				 FOR i:=1 TO gc_ModuleProNo BY 1 DO
						 MEMSET(ADR(tsModuleProcess[i]),0,SIZEOF(tsModuleProcess[i]));
				 END_FOR
			station.iStepAuto:= 20;
  	20://区分上料还是请料
			 IF  station.xEmptying  THEN
					station.iStepAuto:= 1000;
			 ELSIF station.xEmptyDone THEN
					  station.xDone:=TRUE;
						station.iStepAuto:= 0;
			 ELSE
					station.iStepAuto:= 30;
			 END_IF
		30://Restore_after_Estop_Process1-拍照流程
				IF  axBypassSignal[1] OR fbMachine[1].xTryRun THEN
						station.iStepAuto :=110 ;
				ELSE    
						station.iStepAuto :=40; 
				END_IF
		40://启动链板线
			tsModuleProcess[1].xProcessNotStarted:=TRUE;
			IF   NOT _FirstFlag[3] OR station.xSingleRunning THEN
					fbFlowLine.xIRunningPremit:=TRUE;
			END_IF
				station.iStepAuto:=50;	
	 45://
				 fbFlowLine.xIRunningPremit:=TRUE;
				 station.iStepAuto:=46;	
	 46://判断是否需要拍照
				//IF  NOT	_FirstCycle[3] THEN
					 station.iStepAuto:=50;	
				//ELSE
				//	 station.iStepAuto:=80;
				// END_IF
	 50://Y轴去拍照位置
		 arTonDelay[03](IN:=FALSE);
		 fbYAxisMove.xMoveAuto[2]:=TRUE;
		 IF  fbYAxisMove.xMoveInPos[2] THEN
					station.iStepAuto:=60;	
		 END_IF
	60://等待链板线孔板到位 
			arTonDelay[03](IN:=TRUE , PT:=T#10S , Q=> , ET=> ); 
			IF 	fbFlowLine.xQDone  THEN
					 station.iStepAuto:=65;	
			ELSIF fbFlowLine.xQError OR  	arTonDelay[03].Q THEN
			 		arTonDelay[03](IN:=FALSE);
					fbFlowLine.xIInit:=TRUE;
					 station.iStepAuto:=45;	
					station.adwAlarm[1].31	:=	TRUE;//	S01上料工位-链板线运行超时,请复位
			END_IF
	65://链板线停止
				fbFlowLine.xIMotorStop :=TRUE;
			IF NOT  fbFlowLine.xQMotorStart THEN
			 			 station.iStepAuto:=70;	
			END_IF
	70://第一个循环相机拍照
		//tsModuleProcess[1].xProcessStarted:=TRUE;
			Camera.xlTrigger:=TRUE;
			station.iStepAuto:=75;	
	75://相机触发响应
				IF    Camera.xQBusy THEN
						station.iStepAuto:=80;	
				END_IF
	80://等待相机完成且链板线执行完成
			 IF  Camera.xQDone THEN
				 _FirstCycle[3]:=TRUE;
				 station.iStepAuto:=100;		
			 ELSIF  Camera.xQAlarm THEN
					 Camera.xlInit:=TRUE;
					 station.iStepAuto:=70;		
					 station.adwAlarm[1].30	:=	TRUE;//	S01上料工位-相机拍照超时，请检查
			 END_IF
	100://查看相机结果，判断是否料反
		(*位置1*)		
		//tsModuleProcess[1].xProcessCompleted:=TRUE;
		_AlarmDisable:=FALSE;
		FOR  i:=1 TO 4 BY 1 DO
			IF 	sCamera_TO_Plc.iS01Result[i] >=3 THEN
					station.iStepAuto:=101;
					EXIT;
			ELSIF	i =4 THEN
					station.iStepAuto:=110;
			END_IF
		END_FOR
	101://报警,人工处理后重新拍照
		IF  NOT  _AlarmDisable THEN
					IF   sCamera_TO_Plc.iS01Result[1] =3 (*料反*) THEN
						station.adwAlarm[1].01:=TRUE ;//S01链板线上料位置1相机检测到深孔板放反，请检查
					ELSIF  sCamera_TO_Plc.iS01Result[1] =4 (*无料*) THEN
					 	station.adwAlarm[1].26:=TRUE ;//S01链板线上料位置1相机未检测到深孔板，请检查
					END_IF
					IF   sCamera_TO_Plc.iS01Result[2] =3 (*料反*) THEN
						station.adwAlarm[1].02:=TRUE ;//S01链板线上料位置2相机检测到深孔板放反，请检查
					ELSIF  sCamera_TO_Plc.iS01Result[2] =4 (*无料*) THEN
					 	station.adwAlarm[1].27:=TRUE ;//S01链板线上料位置2相机未检到板，请检查
					END_IF	
					IF   sCamera_TO_Plc.iS01Result[3] =3 (*料反*) THEN
 						station.adwAlarm[1].03:= TRUE;//S01链板线上料位置3相机检测到深孔板放反，请检查
					ELSIF  sCamera_TO_Plc.iS01Result[3] =4 (*无料*) THEN
					 	station.adwAlarm[1].28:=TRUE ;//S01链板线上料位置3相机未检到板，请检查
					END_IF
					IF    sCamera_TO_Plc.iS01Result[4] =3 (*料反*) THEN
 						station.adwAlarm[1].04:= TRUE;//S01链板线上料位置4相机检测到深孔板放反，请检查
					ELSIF  sCamera_TO_Plc.iS01Result[4] =4 (*无料*) THEN
					 	station.adwAlarm[1].29:=TRUE ;//S01链板线上料位置4相机未检到板，请检查
					END_IF
					_AlarmDisable:=TRUE;
		END_IF
			station.iStepAuto:=60;
	110://数据传送完成
			tsModuleProcess[1].xQDataCompleted:=TRUE;
			station.iStepAuto:=140;

///预留复检步骤120-140
	140://开始循环。循环次数=2
			bCounter:=1;
			station.iStepAuto :=150; 
	150://循环跳转处
				station.iStepAuto:=160;
	160://Restore_after_Estop_Process2/3 取孔板流程1/2
					station.iStepAuto :=170; 
	170://
			tsModuleProcess[bCounter+1].xProcessNotStarted :=TRUE;
			 station.iStepAuto:=190;		  
	190://XY轴去夹取位置1/2
			fbXAxisMove.xMoveAuto[bCounter +1]:=TRUE;
			fbYAxisMove.xMoveAuto[3]:=TRUE;
			fbClamp_1.aRotateReleaseControl[1]:=TRUE ;
			fbClamp_2.aRotateReleaseControl[1]:=TRUE ;		
			IF fbXAxisMove.xMoveInPos[bCounter+1] AND 
			   fbYAxisMove.xMoveInPos[3] AND 
				 fbClamp_1.xDone AND  
			  fbClamp_2.xDone THEN
					fbClamp_1.xExecute :=FALSE ;
				 fbClamp_2.xExecute :=FALSE ;
				 station.iStepAuto:=200;	
			END_IF
			
	200://Z轴气缸下降
		fbVTCCyl_1.xAuto:=TRUE;
		fbVTCCyl_2.xAuto:=TRUE;
		IF  fbVTCCyl_1.xWP_Delay AND 
			fbVTCCyl_2.xWP_Delay THEN
			 station.iStepAuto:=210;		
		END_IF
	210://电动夹爪夹取
		tsModuleProcess[bCounter+1].xProcessStarted :=TRUE;
		IF  fbmachine[1].xTryRun THEN 
				station.iStepAuto:=215;	
		ELSE
			fbClamp_1.aClampControl[1]:=TRUE;
			fbClamp_2.aClampControl[1]:=TRUE;
			IF (fbClamp_1.xDone OR (fbClamp_1.xGripClampEmpty  AND fbMachine[1].xTryRun)) AND
			 (fbClamp_2.xDone OR (fbClamp_2.xGripClampEmpty  AND fbMachine[1].xTryRun ))   THEN
					fbClamp_1.xExecute :=FALSE ;
					fbClamp_2.xExecute:=FALSE;
					 station.iStepAuto:=215;	
			END_IF
		END_IF
	215://电动夹爪夹取完成
				 tsModuleProcess[bCounter+1].xProcessCompleted :=TRUE;
				 station.iStepAuto:=220;	
	220://Z轴上升
			arClampHavePart[2]:=TRUE;//夹爪2有产品标志位
			
				fbVTCCyl_1.xAuto:=FALSE;
				fbVTCCyl_2.xAuto:=FALSE;
			IF  fbVTCCyl_1.xHP_Delay AND 
				fbVTCCyl_2.xHP_Delay THEN
				 station.iStepAuto:=225;		
			END_IF
	225://判断流程	arClampHavePart[1]:=TRUE;//夹爪1有产品标志位
		
			IF bCounter =2 THEN
					xTakeBoxPremit:=TRUE;//允许链板线执行动作
			END_IF
			station.iStepAuto:=230;	
	230://Restore_after_Estop_Process4 /Process5翻转孔板流程1/2
					station.iStepAuto :=240; 	
	240://判断是否需要翻转
			IF  NOT  fbmachine[1].xTryRun THEN
			 		IF   bCounter =1 THEN
					 			IF 	sCamera_To_Plc.iS01Result[2] =2(*角度反*) OR sCamera_To_Plc.iS01Result[4] =2(*角度反*) THEN 
													 station.iStepAuto:=250;
								ELSE
								 							ariPosNum[1]:=4	;	
															ariPosNum[2]:=4	;	
														 station.iStepAuto:=280;			
								END_IF
								
					ELSIF  bCounter =2 THEN
					 			IF 	sCamera_To_Plc.iS01Result[1] =2(*角度反*) OR sCamera_To_Plc.iS01Result[3] =2(*角度反*) THEN 
													 station.iStepAuto:=250;
								ELSE
								 							ariPosNum[1]:=4	;	
															ariPosNum[2]:=4	;	
														 station.iStepAuto:=280;			
								END_IF
	
					END_IF
			ELSE
			 							station.iStepAuto:=280;			
			END_IF
	250://去翻转位
					tsModuleProcess[bCounter+3].xProcessNotStarted :=TRUE;
			 		 fbXAxisMove.xMoveAuto[6]:=TRUE;
					IF fbXAxisMove.xMoveInPos[6] THEN
						 station.iStepAuto:=260;	
					END_IF 	
  260://空跑
					tsModuleProcess[bCounter+3].xProcessStarted :=TRUE;
					station.iStepAuto:=265;	
	265://夹爪1开始校正
				IF  (sCamera_To_Plc.iS01Result[1] =2(*角度反*) AND bCounter =2 ) OR
						(sCamera_To_Plc.iS01Result[2] =2(*角度反*) AND bCounter =1 ) THEN	
							fbClamp_1.aRotateClampControl[1]:=TRUE ;
							 IF (fbClamp_1.xDone OR (fbClamp_1.xClosecoverFailure AND fbmachine[1].xTryRun)) THEN						
									fbClamp_1.xExecute :=FALSE ;
									station.iStepAuto:= 270;
							END_IF
						ariPosNum[1]:=6	;	
				ELSE
				 		ariPosNum[1]:=4	;	
				 		station.iStepAuto:= 270;
				END_IF
	270://夹爪2开始校正			
				IF  (sCamera_To_Plc.iS01Result[3] =2(*角度反*) AND bCounter =2 ) OR
						(sCamera_To_Plc.iS01Result[4] =2(*角度反*) AND bCounter =1 ) THEN
						fbClamp_2.aRotateClampControl[1]:=TRUE ;
						 IF (fbClamp_2.xDone OR (fbClamp_2.xClosecoverFailure AND fbmachine[1].xTryRun)) THEN			
									fbClamp_2.xExecute :=FALSE ;
									station.iStepAuto:= 280;
							END_IF		
								ariPosNum[2]:=6	;	
				ELSE	
				 				ariPosNum[2]:=4	;	
				 				station.iStepAuto:= 280;
				END_IF	
	280://夹爪矫正完成
			tsModuleProcess[bCounter+3].xProcessCompleted:=TRUE;
			station.iStepAuto:=285;		
	285://检查是否允许放料
			IF  NOT  xLoadingReachedSensor[1]  AND
				NOT  xLoadingReachedSensor[2]  AND 
			(( NOT station.xDone 			   AND
			 (NOT _FirstCycle[4] OR  S08_Mainline.station.xDone)) OR station.xSingleRunning) THEN
				 station.iStepAuto:=290;
				 _FirstCycle[4]:=TRUE;
		  END_IF
	290://X轴放料开始循环计数  =2
			IF ( bXCounter >2) OR NOT _FirstCycle[2] THEN
		 		bXCounter:=1;
				_FirstCycle[2]:=TRUE;
			END_IF
			station.iStepAuto :=291;
	291://是否需要启动链板线
			IF   bCounter  =2 THEN
					fbFlowLine.xIRunningPremit:=TRUE;
			END_IF			
			station.iStepAuto:=295;	
	295://Restore_after_Estop_Process6/7 孔板放料流程1/2
				station.iStepAuto :=300; 
	300://X轴去放料位置	
			tsModuleProcess[bXCounter+5].xProcessNotStarted:=TRUE;
			IF   bXCounter=1 THEN
						fbXAxisMove.xMoveAuto[4]:=TRUE;
						fbYAxisMove.xMoveAuto[ariPosNum[2]]:=TRUE;
								IF fbXAxisMove.xMoveInPos[4] AND 
									 fbYAxisMove.xMoveInPos[ariPosNum[2]] THEN
											 station.iStepAuto:=310;	
								END_IF				
			ELSIF	 bXCounter=2 THEN
			 			 fbXAxisMove.xMoveAuto[5]:=TRUE;
						 fbYAxisMove.xMoveAuto[ariPosNum[1]]:=TRUE;
								IF fbXAxisMove.xMoveInPos[5] AND 
									 fbYAxisMove.xMoveInPos[ariPosNum[1]] THEN
											 station.iStepAuto:=310;
								END_IF				
			END_IF
	//305://同时进行拍照
	//			Camera.xlTrigger:=TRUE;
	//			 station.iStepAuto:=306;
	//306://等待相机触发
	//			IF  Camera.xQBusy THEN
	//			 	station.iStepAuto:=310;
	//		   END_IF
	310://Z轴下降
				IF   bXCounter=1 THEN
						fbVTCCyl_2.xAuto:=TRUE;
						IF fbVTCCyl_2.xWP_Delay THEN
							 station.iStepAuto:=320;	
						END_IF
				ELSIF	 bXCounter=2 THEN
								fbVTCCyl_1.xAuto:=TRUE;
						IF fbVTCCyl_1.xWP_Delay THEN
							 station.iStepAuto:=320;	
						END_IF					
			END_IF
	320://电动夹爪松开
			tsModuleProcess[bXCounter+5].xProcessStarted:=TRUE;
		//	IF  NOT  fbMachine[1].xTryRun THEN
				IF   bXCounter=1 THEN
								fbClamp_2.aReleaseControl[1]:=TRUE;
							IF fbClamp_2.xDone THEN
								fbClamp_2.xExecute:=FALSE;
								 station.iStepAuto:=330;	
							END_IF				
				ELSIF	 bXCounter=2 THEN
							fbClamp_1.aReleaseControl[1]:=TRUE;
							IF fbClamp_1.xDone THEN
								fbClamp_1.xExecute:=FALSE;
								 station.iStepAuto:=330;	
							END_IF			
				END_IF		
		//	ELSE
		//	  	station.iStepAuto:=330;	
		//	 END_IF
	330://传感器检测
				tsModuleProcess[bXCounter+5].xProcessCompleted:=TRUE;
				arClampHavePart[bXCounter]:=FALSE;//夹爪1/2有产品标志位
				IF   xLoadingReachedSensor[bXCounter] OR fbMachine[1].xTryRun THEN
					station.iStepAuto:=340;	
				END_IF
	340://Z轴上升		
				IF   bXCounter=1 THEN
							fbVTCCyl_2.xAuto:=FALSE;
						IF fbVTCCyl_2.xHP_Delay THEN
							 station.iStepAuto:=350;	
						END_IF	
				ELSIF	 bXCounter=2 THEN
							fbVTCCyl_1.xAuto:=FALSE;
						IF fbVTCCyl_1.xHP_Delay THEN
							 station.iStepAuto:=350;	
						END_IF				
				END_IF
	350://Restore_after_Estop_Process8 数据传输流程
			 IF  station.xSingleRunning THEN//OR fbMachine[1].xTryRun THEN
					 station.iStepAuto :=400; 
			ELSIF tsModuleProcess[8].xProcessNotStarted AND NOT  tsModuleProcess[8].xProcessStarted THEN
					 station.iStepAuto :=360; (*process not started*)
			 ELSIF  tsModuleProcess[8].xProcessStarted AND NOT  tsModuleProcess[8].xProcessCompleted THEN
					station.iStepAuto :=370;(*process started*)
			 ELSIF  tsModuleProcess[8].xProcessCompleted AND NOT tsModuleProcess[8].xQDataCompleted  THEN
					 station.iStepAuto :=400 ;(*process completed*)
			 ELSE
					 station.iStepAuto :=360; 
			 END_IF		
		 
	360://任务成功
		 tsModuleProcess[8].xProcessNotStarted:=TRUE;
		 tsModuleProcess[8].xProcessStarted:=TRUE;
		 
		 arProcessDataStation[1].xMaterialOnOff:=TRUE;
		 arProcessDataStation[2].xMaterialOnOff:=TRUE;
		 
		 arProcessDataStation[1].stProduct.xLoading_OK:=TRUE;
		 arProcessDataStation[2].stProduct.xLoading_OK:=TRUE;
			
		 //清空标志位	 
				arProcessDataStation[1].stProduct.xEmptying:=FALSE;
				arProcessDataStation[2].stProduct.xEmptying:=FALSE;		 
		 station.iStepAuto:= 370;
	370://数据unload
			 MEMCPY(ADR(arMainlineFixtureData[arCurFixtureNumStation[1]]),ADR(arProcessDataStation[1]),SIZEOF(arProcessDataStation[1]));
			 MEMCPY(ADR(arMainlineFixtureData[arCurFixtureNumStation[2]]),ADR(arProcessDataStation[2]),SIZEOF(arProcessDataStation[2]));
			 station.iStepAuto:= 380;
	380://本地数据清除
			 	FOR i:=1 TO gc_ModuleProNo BY 1 DO
				 MEMSET(ADR(tsModuleProcess[i]),0,SIZEOF(tsModuleProcess[i]));
			 END_FOR
			 tsModuleProcess[8].xProcessCompleted:=TRUE;
			 station.iStepAuto:= 400;		
			 
			
	400://放料完成
			IF bXCounter =2 THEN
				station.xDone:=TRUE;
			END_IF
			station.iStepAuto:=420;
	420://X轴循环+1
			bXCounter :=bXCounter +1;
			station.iStepAuto:=430;	

	430:  
		IF   bXCounter<=2 THEN
				station.iStepAuto:=295;	
		ELSE
				station.iStepAuto:=440;	
		END_IF

	440://循环+1
			bCounter :=bCounter +1;
			 station.iStepAuto:=450;
	450://
		IF   bCounter <=2  THEN 
		 	  station.iStepAuto:=150;
		ELSIF	 bCounter >2 THEN
		 		station.iStepAuto:=999;
		END_IF
		
	999://----Single Run Finish----
		station.iStepAuto :=0;
		station.xSingleRunFlag:=FALSE;
		station.xCycleEnable:=FALSE;	
	//	station.xDone:=TRUE;
{region "请料程序"}
	1000://进入请料流程
		 		//写入数据
			 	arProcessDataStation[1].xMaterialOnOff:=FALSE;
		 		arProcessDataStation[2].xMaterialOnOff:=FALSE;
				arProcessDataStation[1].stProduct.xLoading_OK:=FALSE;
			  arProcessDataStation[2].stProduct.xLoading_OK:=FALSE;
				//清空标志位	 
				arProcessDataStation[1].stProduct.xEmptying:=TRUE;
				arProcessDataStation[2].stProduct.xEmptying:=TRUE;
			 MEMCPY(ADR(arMainlineFixtureData[arCurFixtureNumStation[1]]),ADR(arProcessDataStation[1]),SIZEOF(arProcessDataStation[1]));
			 MEMCPY(ADR(arMainlineFixtureData[arCurFixtureNumStation[2]]),ADR(arProcessDataStation[2]),SIZEOF(arProcessDataStation[2]));
			 station.iStepAuto :=1010;
	1010://允许主流线前进
					
		 		station.xDone:=TRUE;
				station.iStepAuto :=1020;
	1020://伺服去待机位置
			 fbXAxisMove.xMoveAuto[1]:=TRUE;
			 fbYAxisMove.xMoveAuto[1]:=TRUE;
			IF fbXAxisMove.xMoveInPos[1] AND 
				 fbYAxisMove.xMoveInPos[1]  THEN
				station.iStepAuto:=1030;	
			END_IF
  1030://电动夹爪初始化
				 fbClamp_1.xInitControl:=TRUE ;
					fbClamp_2.xInitControl:=TRUE ;
				IF  fbClamp_1.xDone   AND
						fbClamp_2.xDone  THEN 
						 fbClamp_1.xExecute :=FALSE;
						 fbClamp_2.xExecute:=FALSE;
						 station.iStepAuto:=1040;
				END_IF				
  1040://电动夹爪去初始位置
						 fbClamp_1.aReleaseControl[1]:=TRUE ;
						 fbClamp_2.aReleaseControl[1]:=TRUE ;
					IF  fbClamp_1.xDone AND
							fbClamp_2.xDone THEN 
								fbClamp_1.xExecute :=FALSE;
								fbClamp_2.xExecute:=FALSE;
								 station.iStepAuto:=1050;
					END_IF						
	1050://链板线初始化
					 fbFlowLine.xIInit:=TRUE;
					 station.iStepAuto:=1060;
  1060://等待完成
					IF  NOT fbFlowLine.xQBusy THEN
							station.iStepAuto:=1100;
					END_IF
	1100://当站清料完成
			 		 station.xEmptying:=FALSE;
			 		 station.xEmptyDone:=TRUE;
					 station.iStepAuto:=0;				
{endregion}
	
	
	
	ELSE
		;	
END_CASE

END_IF
END_ACTION

ACTION FlowAuto_1:

//-----------------------------------------初始化是否完成判断----------------------------------------------
IF NOT station.xInitDone THEN
 	station.iStepAuto:=0;
 	station.xDone:=FALSE;
ELSIF station.xRunning  OR 
//(tsModuleProcess[1].xProcessStarted AND  NOT tsModuleProcess[1].xProcessCompleted)  OR//相机拍照流程
(	tsModuleProcess[bCounter+1].xProcessStarted AND  NOT tsModuleProcess[bCounter+1].xProcessCompleted)  OR //电动夹爪夹取流程
(tsModuleProcess[bCounter+3].xProcessStarted AND  NOT tsModuleProcess[bCounter+3].xProcessCompleted)  OR //孔板翻转流程流程
(	tsModuleProcess[bXCounter+5].xProcessStarted AND NOT 	tsModuleProcess[bXCounter+5].xProcessCompleted) //电动夹爪松开流程
THEN
//-----------------------------------------动作步骤--------------------------------------------------------
CASE station.iStepAuto OF	  
	0: //----Home Step，等待启动----
		IF station.xDisabled 
			AND station.xCanRun 
			AND NOT fbMachine[1].xStopped 
			AND NOT station.xSingleRunning 
		THEN
			station.xDone:=TRUE;
		END_IF
		IF  station.xSingleRunning 
			OR station.xCanRun 
			//AND NOT station.xDone 
			AND NOT station.xDisabled 
			AND NOT fbMachine[1].xStopped
		THEN
			station.xCycleEnable:=TRUE;
			//station.xDone:= FALSE;  
			station.iStepAuto:= 10;
		END_IF
	10://复位
			Camera.xlInit:=TRUE;
			FOR  i:=1 TO  4 BY  1 DO
		 		sCamera_To_Plc.iS01Result[i]:=0;
			END_FOR
			MEMSET(ADR(arProcessDataStation[1]),0,SIZEOF(arProcessDataStation[1]));
			MEMSET(ADR(arProcessDataStation[2]),0,SIZEOF(arProcessDataStation[2]));
		
				 FOR i:=1 TO gc_ModuleProNo BY 1 DO
						 MEMSET(ADR(tsModuleProcess[i]),0,SIZEOF(tsModuleProcess[i]));
				 END_FOR
			station.iStepAuto:= 20;
  	20://区分上料还是请料
			 IF  station.xEmptying  THEN
					station.iStepAuto:= 1000;
			 ELSIF station.xEmptyDone THEN
					  station.xDone:=TRUE;
						station.iStepAuto:= 0;
			 ELSE
					station.iStepAuto:= 30;
			 END_IF
		30://Restore_after_Estop_Process1-拍照流程
				IF  axBypassSignal[1] OR fbMachine[1].xTryRun THEN
						station.iStepAuto :=110 ;
				ELSE    
						station.iStepAuto :=40; 
				END_IF
		40://启动链板线
			tsModuleProcess[1].xProcessNotStarted:=TRUE;
			IF   NOT _FirstFlag[3] OR station.xSingleRunning THEN
					fbFlowLine.xIRunningPremit:=TRUE;
			END_IF
				station.iStepAuto:=50;	
	 45://
				 fbFlowLine.xIRunningPremit:=TRUE;
				 station.iStepAuto:=46;	
	 46://判断是否需要拍照
				//IF  NOT	_FirstCycle[3] THEN
					 station.iStepAuto:=50;	
				//ELSE
				//	 station.iStepAuto:=80;
				// END_IF
	 50://Y轴去拍照位置
		 arTonDelay[03](IN:=FALSE);
		 fbYAxisMove.xMoveAuto[2]:=TRUE;
		 IF  fbYAxisMove.xMoveInPos[2] THEN
					station.iStepAuto:=60;	
		 END_IF
	60://等待链板线孔板到位 
			arTonDelay[03](IN:=TRUE , PT:=T#10S , Q=> , ET=> ); 
			IF 	fbFlowLine.xQDone  THEN
					 station.iStepAuto:=65;	
			ELSIF fbFlowLine.xQError OR  	arTonDelay[03].Q THEN
			 		arTonDelay[03](IN:=FALSE);
					fbFlowLine.xIInit:=TRUE;
					 station.iStepAuto:=45;	
					station.adwAlarm[1].31	:=	TRUE;//	S01上料工位-链板线运行超时,请复位
			END_IF
	65://链板线停止
				fbFlowLine.xIMotorStop :=TRUE;
			IF NOT  fbFlowLine.xQMotorStart THEN
			 			 station.iStepAuto:=70;	
			END_IF
	70://第一个循环相机拍照
		//tsModuleProcess[1].xProcessStarted:=TRUE;
			Camera.xlTrigger:=TRUE;
			station.iStepAuto:=75;	
	75://相机触发响应
				IF    Camera.xQBusy THEN
						station.iStepAuto:=80;	
				END_IF
	80://等待相机完成且链板线执行完成
			 IF  Camera.xQDone THEN
				 _FirstCycle[3]:=TRUE;
				 station.iStepAuto:=100;		
			 ELSIF  Camera.xQAlarm THEN
					 Camera.xlInit:=TRUE;
					 station.iStepAuto:=70;		
					 station.adwAlarm[1].30	:=	TRUE;//	S01上料工位-相机拍照超时，请检查
			 END_IF
	100://查看相机结果，判断是否料反
		(*位置1*)		
		//tsModuleProcess[1].xProcessCompleted:=TRUE;
		_AlarmDisable:=FALSE;
		FOR  i:=1 TO 4 BY 1 DO
			IF 	sCamera_TO_Plc.iS01Result[i] >=3 THEN
					station.iStepAuto:=101;
					EXIT;
			ELSIF	i =4 THEN
					station.iStepAuto:=110;
			END_IF
		END_FOR
	101://报警,人工处理后重新拍照
		IF  NOT  _AlarmDisable THEN
					IF   sCamera_TO_Plc.iS01Result[1] =3 (*料反*) THEN
						station.adwAlarm[1].01:=TRUE ;//S01链板线上料位置1相机检测到深孔板放反，请检查
					ELSIF  sCamera_TO_Plc.iS01Result[1] =4 (*无料*) THEN
					 	station.adwAlarm[1].26:=TRUE ;//S01链板线上料位置1相机未检测到深孔板，请检查
					END_IF
					IF   sCamera_TO_Plc.iS01Result[2] =3 (*料反*) THEN
						station.adwAlarm[1].02:=TRUE ;//S01链板线上料位置2相机检测到深孔板放反，请检查
					ELSIF  sCamera_TO_Plc.iS01Result[2] =4 (*无料*) THEN
					 	station.adwAlarm[1].27:=TRUE ;//S01链板线上料位置2相机未检到板，请检查
					END_IF	
					IF   sCamera_TO_Plc.iS01Result[3] =3 (*料反*) THEN
 						station.adwAlarm[1].03:= TRUE;//S01链板线上料位置3相机检测到深孔板放反，请检查
					ELSIF  sCamera_TO_Plc.iS01Result[3] =4 (*无料*) THEN
					 	station.adwAlarm[1].28:=TRUE ;//S01链板线上料位置3相机未检到板，请检查
					END_IF
					IF    sCamera_TO_Plc.iS01Result[4] =3 (*料反*) THEN
 						station.adwAlarm[1].04:= TRUE;//S01链板线上料位置4相机检测到深孔板放反，请检查
					ELSIF  sCamera_TO_Plc.iS01Result[4] =4 (*无料*) THEN
					 	station.adwAlarm[1].29:=TRUE ;//S01链板线上料位置4相机未检到板，请检查
					END_IF
					_AlarmDisable:=TRUE;
		END_IF
			station.iStepAuto:=60;
	110://数据传送完成
			tsModuleProcess[1].xQDataCompleted:=TRUE;
			station.iStepAuto:=140;

///预留复检步骤120-140
	140://开始循环。循环次数=2
			bCounter:=1;
			bXCounter:=1;
			station.iStepAuto :=150; 
	150://循环跳转处
				station.iStepAuto:=160;
	160://Restore_after_Estop_Process2/3 取孔板流程1/2
					station.iStepAuto :=170; 
	170://
			tsModuleProcess[bCounter+1].xProcessNotStarted :=TRUE;
			 station.iStepAuto:=190;		  
	190://XY轴去夹取位置1/2
			fbXAxisMove.xMoveAuto[bCounter +1]:=TRUE;
			fbYAxisMove.xMoveAuto[3]:=TRUE;
			ERG_20C_1.stDeviceOpe.aRotateReleaseControl[1]:=TRUE ;
			ERG_20C_2.stDeviceOpe.aRotateReleaseControl[1]:=TRUE ;	
			IF    ERG_20C_1.stDevice.xQBusy AND 
			 			ERG_20C_2.stDevice.xQBusy THEN
						 station.iStepAuto:=195;	
			END_IF
	195://等待
			IF fbXAxisMove.xMoveInPos[bCounter+1] AND 
			   fbYAxisMove.xMoveInPos[3] AND 
				 ERG_20C_1.stDevice.xQDone AND  
			   ERG_20C_2.stDevice.xQDone THEN
				 station.iStepAuto:=200;	
			END_IF
	200://Z轴气缸下降
		fbVTCCyl_1.xAuto:=TRUE;
		fbVTCCyl_2.xAuto:=TRUE;
		IF  fbVTCCyl_1.xWP_Delay AND 
			fbVTCCyl_2.xWP_Delay THEN
			 station.iStepAuto:=210;		
		END_IF
	210://电动夹爪夹取
			tsModuleProcess[bCounter+1].xProcessStarted :=TRUE;
			ERG_20C_1.stDeviceOpe.aClampControl[1]:=TRUE;
			ERG_20C_2.stDeviceOpe.aClampControl[1]:=TRUE;  
			IF    ERG_20C_1.stDevice.xQBusy AND 
			 			ERG_20C_2.stDevice.xQBusy THEN
						 station.iStepAuto:=215;	
			END_IF
		
	215://电动夹爪夹取完成
				 IF ERG_20C_1.stDevice.xQDone AND 
			 			ERG_20C_2.stDevice.xQDone THEN
						 tsModuleProcess[bCounter+1].xProcessCompleted :=TRUE;
						 station.iStepAuto:=220;	
			END_IF
	220://Z轴上升
			arClampHavePart[2]:=TRUE;//夹爪2有产品标志位
			
				fbVTCCyl_1.xAuto:=FALSE;
				fbVTCCyl_2.xAuto:=FALSE;
			IF  fbVTCCyl_1.xHP_Delay AND 
				fbVTCCyl_2.xHP_Delay THEN
				 station.iStepAuto:=225;		
			END_IF
	225://判断流程	arClampHavePart[1]:=TRUE;//夹爪1有产品标志位
		
			IF bCounter =2 THEN
					xTakeBoxPremit:=TRUE;//允许链板线执行动作
			END_IF
			station.iStepAuto:=230;	
	230://Restore_after_Estop_Process4 /Process5翻转孔板流程1/2
					station.iStepAuto :=240; 	
	240://判断是否需要翻转
			IF  NOT  fbmachine[1].xTryRun THEN
			 		IF   bCounter =1 THEN
					 			IF 	sCamera_To_Plc.iS01Result[2] =2(*角度反*) OR sCamera_To_Plc.iS01Result[4] =2(*角度反*) THEN 
													 station.iStepAuto:=250;
								ELSE
								 							ariPosNum[1]:=4	;	
															ariPosNum[2]:=4	;	
														 station.iStepAuto:=280;			
								END_IF
								
					ELSIF  bCounter =2 THEN
					 			IF 	sCamera_To_Plc.iS01Result[1] =2(*角度反*) OR sCamera_To_Plc.iS01Result[3] =2(*角度反*) THEN 
													 station.iStepAuto:=250;
								ELSE
								 							ariPosNum[1]:=4	;	
															ariPosNum[2]:=4	;	
														 station.iStepAuto:=280;			
								END_IF
	
					END_IF
			ELSE
			 							station.iStepAuto:=280;			
			END_IF
	250://去翻转位
					tsModuleProcess[bCounter+3].xProcessNotStarted :=TRUE;
			 		 fbXAxisMove.xMoveAuto[6]:=TRUE;
					IF fbXAxisMove.xMoveInPos[6] THEN
						 station.iStepAuto:=260;	
					END_IF 	
  260://空跑
					tsModuleProcess[bCounter+3].xProcessStarted :=TRUE;
					station.iStepAuto:=265;	
	265://夹爪1开始校正
				IF  (sCamera_To_Plc.iS01Result[1] =2(*角度反*) AND bCounter =2 ) OR
						(sCamera_To_Plc.iS01Result[2] =2(*角度反*) AND bCounter =1 ) THEN	
								ERG_20C_1.stDeviceOpe.aRotateClampControl[1]:=TRUE ;
							 IF ERG_20C_1.stDevice.xQBusy  THEN					
									station.iStepAuto:= 266;
							END_IF
						ariPosNum[1]:=6	;	
				ELSE
				 		ariPosNum[1]:=4	;	
				 		station.iStepAuto:= 270;
				END_IF
	266://
				IF ERG_20C_1.stDevice.xQDone  THEN					
									station.iStepAuto:= 270;
				END_IF
	270://夹爪2开始校正			
				IF  (sCamera_To_Plc.iS01Result[3] =2(*角度反*) AND bCounter =2 ) OR
						(sCamera_To_Plc.iS01Result[4] =2(*角度反*) AND bCounter =1 ) THEN
							ERG_20C_2.stDeviceOpe.aRotateClampControl[1]:=TRUE ;
							 IF ERG_20C_2.stDevice.xQBusy  THEN					
									station.iStepAuto:= 275;
							END_IF
								ariPosNum[2]:=6	;	
				ELSE	
				 				ariPosNum[2]:=4	;	
				 				station.iStepAuto:= 280;
				END_IF	
  275://
				IF ERG_20C_2.stDevice.xQDone  THEN					
							station.iStepAuto:= 280;
				END_IF
	280://夹爪矫正完成
			tsModuleProcess[bCounter+3].xProcessCompleted:=TRUE;
			station.iStepAuto:=285;		
	285://检查是否允许放料
			IF  NOT  xLoadingReachedSensor[1]  AND
				NOT  xLoadingReachedSensor[2]  AND 
			(( NOT station.xDone 			   AND
			 (NOT _FirstCycle[4] OR  S08_Mainline.station.xDone)) OR station.xSingleRunning) THEN
				 station.iStepAuto:=290;
				 _FirstCycle[4]:=TRUE;
		  END_IF
	290://X轴放料开始循环计数  =2
			IF ( bXCounter >2) OR NOT _FirstCycle[2] THEN
		 		bXCounter:=1;
				_FirstCycle[2]:=TRUE;
			END_IF
			station.iStepAuto :=291;
	291://是否需要启动链板线
			IF   bCounter  =2 THEN
					fbFlowLine.xIRunningPremit:=TRUE;
			END_IF			
			station.iStepAuto:=295;	
	295://Restore_after_Estop_Process6/7 孔板放料流程1/2
				station.iStepAuto :=300; 
	300://X轴去放料位置	
			tsModuleProcess[bXCounter+5].xProcessNotStarted:=TRUE;
			IF   bXCounter=1 THEN
						fbXAxisMove.xMoveAuto[4]:=TRUE;
						fbYAxisMove.xMoveAuto[ariPosNum[2]]:=TRUE;
								IF fbXAxisMove.xMoveInPos[4] AND 
									 fbYAxisMove.xMoveInPos[ariPosNum[2]] THEN
											 station.iStepAuto:=310;	
								END_IF				
			ELSIF	 bXCounter=2 THEN
			 			 fbXAxisMove.xMoveAuto[5]:=TRUE;
						 fbYAxisMove.xMoveAuto[ariPosNum[1]]:=TRUE;
								IF fbXAxisMove.xMoveInPos[5] AND 
									 fbYAxisMove.xMoveInPos[ariPosNum[1]] THEN
											 station.iStepAuto:=310;
								END_IF				
			END_IF
	//305://同时进行拍照
	//			Camera.xlTrigger:=TRUE;
	//			 station.iStepAuto:=306;
	//306://等待相机触发
	//			IF  Camera.xQBusy THEN
	//			 	station.iStepAuto:=310;
	//		   END_IF
	310://Z轴下降
				IF   bXCounter=1 THEN
						fbVTCCyl_2.xAuto:=TRUE;
						IF fbVTCCyl_2.xWP_Delay THEN
							 station.iStepAuto:=320;	
						END_IF
				ELSIF	 bXCounter=2 THEN
								fbVTCCyl_1.xAuto:=TRUE;
						IF fbVTCCyl_1.xWP_Delay THEN
							 station.iStepAuto:=320;	
						END_IF					
			END_IF
	320://电动夹爪松开
			tsModuleProcess[bXCounter+5].xProcessStarted:=TRUE;
				IF   bXCounter=1 THEN
								ERG_20C_2.stDeviceOpe.aReleaseControl[1]:=TRUE;
							IF ERG_20C_2.stDevice.xQBusy  THEN
								 station.iStepAuto:=325;	
							END_IF				
				ELSIF	 bXCounter=2 THEN
							ERG_20C_1.stDeviceOpe.aReleaseControl[1]:=TRUE;
							IF ERG_20C_1.stDevice.xQBusy  THEN
								 station.iStepAuto:=326;	
							END_IF		
				END_IF		
	325: //等待夹爪动作完成
				 IF ERG_20C_2.stDevice.xQDone  THEN
								 station.iStepAuto:=330;	
				 END_IF			
	326: //等待夹爪动作完成
				 IF ERG_20C_1.stDevice.xQDone  THEN
								 station.iStepAuto:=330;	
				 END_IF		  	
	330://传感器检测
				tsModuleProcess[bXCounter+5].xProcessCompleted:=TRUE;
				arClampHavePart[bXCounter]:=FALSE;//夹爪1/2有产品标志位
				IF   xLoadingReachedSensor[bXCounter] OR fbMachine[1].xTryRun THEN
					station.iStepAuto:=340;	
				END_IF
	340://Z轴上升		
				IF   bXCounter=1 THEN
							fbVTCCyl_2.xAuto:=FALSE;
						IF fbVTCCyl_2.xHP_Delay THEN
							 station.iStepAuto:=350;	
						END_IF	
				ELSIF	 bXCounter=2 THEN
							fbVTCCyl_1.xAuto:=FALSE;
						IF fbVTCCyl_1.xHP_Delay THEN
							 station.iStepAuto:=350;	
						END_IF				
				END_IF
	350://Restore_after_Estop_Process8 数据传输流程
			 IF  station.xSingleRunning THEN//OR fbMachine[1].xTryRun THEN
					 station.iStepAuto :=400; 
			ELSIF tsModuleProcess[8].xProcessNotStarted AND NOT  tsModuleProcess[8].xProcessStarted THEN
					 station.iStepAuto :=360; (*process not started*)
			 ELSIF  tsModuleProcess[8].xProcessStarted AND NOT  tsModuleProcess[8].xProcessCompleted THEN
					station.iStepAuto :=370;(*process started*)
			 ELSIF  tsModuleProcess[8].xProcessCompleted AND NOT tsModuleProcess[8].xQDataCompleted  THEN
					 station.iStepAuto :=400 ;(*process completed*)
			 ELSE
					 station.iStepAuto :=360; 
			 END_IF		
		 
	360://任务成功
		 tsModuleProcess[8].xProcessNotStarted:=TRUE;
		 tsModuleProcess[8].xProcessStarted:=TRUE;
		 
		 arProcessDataStation[1].xMaterialOnOff:=TRUE;
		 arProcessDataStation[2].xMaterialOnOff:=TRUE;
		 
		 arProcessDataStation[1].stProduct.xLoading_OK:=TRUE;
		 arProcessDataStation[2].stProduct.xLoading_OK:=TRUE;
			
		 //清空标志位	 
				arProcessDataStation[1].stProduct.xEmptying:=FALSE;
				arProcessDataStation[2].stProduct.xEmptying:=FALSE;		 
		 station.iStepAuto:= 370;
	370://数据unload
			 MEMCPY(ADR(arMainlineFixtureData[arCurFixtureNumStation[1]]),ADR(arProcessDataStation[1]),SIZEOF(arProcessDataStation[1]));
			 MEMCPY(ADR(arMainlineFixtureData[arCurFixtureNumStation[2]]),ADR(arProcessDataStation[2]),SIZEOF(arProcessDataStation[2]));
			 station.iStepAuto:= 380;
	380://本地数据清除
			 	FOR i:=1 TO gc_ModuleProNo BY 1 DO
				 MEMSET(ADR(tsModuleProcess[i]),0,SIZEOF(tsModuleProcess[i]));
			 END_FOR
			 tsModuleProcess[8].xProcessCompleted:=TRUE;
			 station.iStepAuto:= 400;		
			 
			
	400://放料完成
			IF bXCounter =2 THEN
				station.xDone:=TRUE;
			END_IF
			station.iStepAuto:=420;
	420://X轴循环+1
			bXCounter :=bXCounter +1;
			station.iStepAuto:=430;	

	430:  
		IF   bXCounter<=2 THEN
				station.iStepAuto:=295;	
		ELSE
				station.iStepAuto:=440;	
		END_IF

	440://循环+1
			bCounter :=bCounter +1;
			 station.iStepAuto:=450;
	450://
		IF   bCounter <=2  THEN 
		 	  station.iStepAuto:=150;
		ELSIF	 bCounter >2 THEN
		 		station.iStepAuto:=999;
		END_IF
		
	999://----Single Run Finish----
		station.iStepAuto :=0;
		station.xSingleRunFlag:=FALSE;
		station.xCycleEnable:=FALSE;	
	//	station.xDone:=TRUE;
{region "请料程序"}
	1000://进入请料流程
		 		//写入数据
			 	arProcessDataStation[1].xMaterialOnOff:=FALSE;
		 		arProcessDataStation[2].xMaterialOnOff:=FALSE;
				arProcessDataStation[1].stProduct.xLoading_OK:=FALSE;
			  arProcessDataStation[2].stProduct.xLoading_OK:=FALSE;
				//清空标志位	 
				arProcessDataStation[1].stProduct.xEmptying:=TRUE;
				arProcessDataStation[2].stProduct.xEmptying:=TRUE;
			 MEMCPY(ADR(arMainlineFixtureData[arCurFixtureNumStation[1]]),ADR(arProcessDataStation[1]),SIZEOF(arProcessDataStation[1]));
			 MEMCPY(ADR(arMainlineFixtureData[arCurFixtureNumStation[2]]),ADR(arProcessDataStation[2]),SIZEOF(arProcessDataStation[2]));
			 station.iStepAuto :=1010;
	1010://允许主流线前进
					
		 		station.xDone:=TRUE;
				station.iStepAuto :=1020;
	1020://伺服去待机位置
			 fbXAxisMove.xMoveAuto[1]:=TRUE;
			 fbYAxisMove.xMoveAuto[1]:=TRUE;
			IF fbXAxisMove.xMoveInPos[1] AND 
				 fbYAxisMove.xMoveInPos[1]  THEN
				station.iStepAuto:=1030;	
			END_IF
	1030://电动夹爪初始化
					ERG_20C_1.stDeviceOpe.xInitControl:=TRUE;
					ERG_20C_2.stDeviceOpe.xInitControl:=TRUE;
		 		IF   ERG_20C_1.stDevice.xQBusy AND  ERG_20C_2.stDevice.xQBusy THEN
				 				station.iStepAuto:=1040;		
				END_IF
 1040://等待夹爪初始化完成
				 IF     ERG_20C_1.stDevice.xQDone AND 
								ERG_20C_2.stDevice.xQDone THEN
								station.iStepAuto:=1050;	
				 END_IF
 1050://电动夹爪去打开位置
					 ERG_20C_1.stDeviceOpe.aReleaseControl[1]:=TRUE;
					 ERG_20C_2.stDeviceOpe.aReleaseControl[1]:=TRUE;
				 IF   ERG_20C_1.stDevice.xQBusy AND  ERG_20C_2.stDevice.xQBusy THEN
								 station.iStepAuto:=1060;	
				 END_IF	
 1060://等待夹爪初始化完成
				 IF     ERG_20C_1.stDevice.xQDone AND 
								ERG_20C_2.stDevice.xQDone THEN
								station.iStepAuto:=1070;	
				 END_IF
	1070://链板线初始化
					 fbFlowLine.xIInit:=TRUE;
					 station.iStepAuto:=1080;
  1080://等待完成
					IF  NOT fbFlowLine.xQBusy THEN
							station.iStepAuto:=1100;
					END_IF
	1100://当站清料完成
			 		 station.xEmptying:=FALSE;
			 		 station.xEmptyDone:=TRUE;
					 station.iStepAuto:=0;				
{endregion}
	
	
	
	ELSE
		;	
END_CASE

END_IF
END_ACTION

ACTION FlowInit:
IF NOT station.xIniting THEN
  station.iStepInit:=0;    

ELSE
//--------------------------------------------初始化步序----------------------------------
CASE station.iStepInit OF	
 0://  
  	IF station.xIniting THEN	
  	  station.iStepInit:=10;	
  	END_IF	
10://复位数据
		FOR i:=1 TO gc_ModuleProNo BY 1 DO
				MEMSET(ADR(tsModuleProcess[i]),0,SIZEOF(tsModuleProcess[i]));
		END_FOR
		FOR  i:=1 TO  4 BY  1 DO
		 		sCamera_To_Plc.iS01Result[i]:=0;
		END_FOR
		fbClamp_1.xInitControl:=FALSE;
		fbClamp_1.xInitControl:=FALSE ;
		fbClamp_1.aRotateClampControl[1]:=FALSE ;
		fbClamp_2.aRotateClampControl[1]:=FALSE ;
		fbClamp_1.xExecute :=FALSE;
		fbClamp_2.xExecute:=FALSE;
		IF NOT fbMachine[1].xTryRun THEN
				Camera.xlInit:=TRUE;
		END_IF
    station.iStepInit := 20;
20://Z轴上升
	 fbVTCCyl_1.xinit := TRUE; 
	 fbVTCCyl_2.xInit:=TRUE;
	IF fbVTCCyl_1.xHP_Delay AND fbVTCCyl_2.xHP_Delay  THEN
    		station.iStepInit:=40;	
	END_IF		
40: //伺服上电
  	 fbXAxisMove.xPowerInit := TRUE ;
	 fbYAxisMove.xPowerInit := TRUE ;
	IF fbXAxisMove.xPowerOn AND   fbYAxisMove.xPowerOn THEN 
    	station.iStepInit:=50;	
	END_IF
50://伺服去待机位置
		fbXAxisMove.xMoveAuto[1]:=TRUE;
		fbYAxisMove.xMoveAuto[1]:=TRUE;
		IF fbXAxisMove.xMoveInPos[1] AND fbYAxisMove.xMoveInPos[1]  THEN
			station.iStepInit:=60;	
		END_IF
60://电动夹爪初始化
				 fbClamp_1.xInitControl:=TRUE ;
				 fbClamp_2.xInitControl:=TRUE ;
		 IF  fbClamp_1.xDone   AND  fbClamp_2.xDone  THEN 
			fbClamp_1.xExecute :=FALSE;
			fbClamp_2.xExecute:=FALSE;
			station.iStepInit:=70;
		 END_IF				
70://电动夹爪去初始位置
				fbClamp_1.aReleaseControl[1]:=TRUE ;
				fbClamp_2.aReleaseControl[1]:=TRUE ;
		 IF  fbClamp_1.xDone AND fbClamp_2.xDone THEN 
			fbClamp_1.xExecute :=FALSE;
			fbClamp_2.xExecute:=FALSE;
			station.iStepInit:=80;
		 END_IF						
80://链板线初始化
		fbFlowLine.xIInit:=TRUE;
		station.iStepInit:=90;
90://等待完成
		IF  NOT fbFlowLine.xQBusy THEN
			 	station.iStepInit:=100;
		END_IF
100://
       station.iStepInit:=999;	

999://初始化完成	
	station.iStepInit:=0;
	station.xInitDone:=TRUE;  
END_CASE
END_IF
END_ACTION

ACTION FlowInit_1:
IF NOT station.xIniting THEN
  station.iStepInit:=0;    

ELSE
//--------------------------------------------初始化步序----------------------------------
CASE station.iStepInit OF	
 0://  
  	IF station.xIniting THEN	
  	  station.iStepInit:=10;	
  	END_IF	
10://复位数据
		FOR i:=1 TO gc_ModuleProNo BY 1 DO
				MEMSET(ADR(tsModuleProcess[i]),0,SIZEOF(tsModuleProcess[i]));
		END_FOR
		FOR  i:=1 TO  4 BY  1 DO
		 		sCamera_To_Plc.iS01Result[i]:=0;
		END_FOR
		fbClamp_1.xInitControl:=FALSE;
		fbClamp_1.xInitControl:=FALSE ;
		fbClamp_1.aRotateClampControl[1]:=FALSE ;
		fbClamp_2.aRotateClampControl[1]:=FALSE ;
		fbClamp_1.xExecute :=FALSE;
		fbClamp_2.xExecute:=FALSE;
		IF NOT fbMachine[1].xTryRun THEN
				Camera.xlInit:=TRUE;
		END_IF
    station.iStepInit := 20;
20://Z轴上升
	 fbVTCCyl_1.xinit := TRUE; 
	 fbVTCCyl_2.xInit:=TRUE;
	IF fbVTCCyl_1.xHP_Delay AND fbVTCCyl_2.xHP_Delay  THEN
    		station.iStepInit:=40;	
	END_IF		
40: //伺服上电
  	 fbXAxisMove.xPowerInit := TRUE ;
	 fbYAxisMove.xPowerInit := TRUE ;
	IF fbXAxisMove.xPowerOn AND   fbYAxisMove.xPowerOn THEN 
    	station.iStepInit:=50;	
	END_IF
50://伺服去待机位置
		fbXAxisMove.xMoveAuto[1]:=TRUE;
		fbYAxisMove.xMoveAuto[1]:=TRUE;
		IF fbXAxisMove.xMoveInPos[1] AND fbYAxisMove.xMoveInPos[1]  THEN
			station.iStepInit:=60;	
		END_IF
60://电动夹爪初始化
					ERG_20C_1.stDeviceOpe.xInitControl:=TRUE;
					ERG_20C_2.stDeviceOpe.xInitControl:=TRUE;
		 		IF   ERG_20C_1.stDevice.xQBusy AND  ERG_20C_2.stDevice.xQBusy THEN
				 				station.iStepInit:=65;		
				END_IF
65://等待夹爪初始化完成
				IF     ERG_20C_1.stDevice.xQDone AND 
				 			 ERG_20C_2.stDevice.xQDone THEN
							 	station.iStepInit:=70;
				END_IF
70://电动夹爪去打开位置
					ERG_20C_1.stDeviceOpe.aReleaseControl[1]:=TRUE;
					ERG_20C_2.stDeviceOpe.aReleaseControl[1]:=TRUE;
		 		IF   ERG_20C_1.stDevice.xQBusy AND  ERG_20C_2.stDevice.xQBusy THEN
				 				station.iStepInit:=75;		
				END_IF	
75://等待夹爪初始化完成
			  IF     ERG_20C_1.stDevice.xQDone AND 
				 			 ERG_20C_2.stDevice.xQDone THEN
							 	station.iStepInit:=80;
				END_IF
80://链板线初始化
		fbFlowLine.xIInit:=TRUE;
		station.iStepInit:=90;
90://等待完成
		IF  NOT fbFlowLine.xQBusy THEN
			 	station.iStepInit:=100;
		END_IF
100://
       station.iStepInit:=999;	

999://初始化完成	
	station.iStepInit:=0;
	station.xInitDone:=TRUE;  
END_CASE
END_IF
END_ACTION

ACTION FlowLine:
	
	fbFlowLine(
	arIReachedSensor:= arFlowLineReachedSensor,
	arIVTCCylHPSensor:=arVTCPressCylHPSensor , 
	arIVTCCylWPSensor:=arVTCPressCylWPSensor , 
	xIRunningPremit:= ,
	xIInit:= ,//station.xIniting,
	xIEmptyDone:=  fbMachine[1].xEmptyDone, 
	xITryRun:= fbMachine[1].xTryRun, 
	xIMotorEstop:=  not  fbMachine[1].xEStop, 
	xIMotorStartButtonHmi:=arFlowLineControl[1] , 
	xIMotorStopButtonHmi:= arFlowLineControl[2], 
	xIManualMode:= fbMachine[1].xManualMode , 
	xIAutoMode	:= fbMachine[1].xAutoMode, 
	xIDeviceRunning:=TRUE,
	arQVTCCylHPValve=> , 
	arQVTCCylWPValve=> , 
	xQMotorEstop=> QxFlowLineSpeedCtrl_1, 
	xQMotorStop=> QxFlowLineStop, 
	xQMotorStart=>QxFlowLineStart , 
	xQBusy=> , 
	xQError=> );
END_ACTION

ACTION General:
MachineInitR_TRIG(CLK:=fbMachine[1].xInitDone OR fbMachine[1].xEmptyDone , Q=> );
IF  MachineInitR_TRIG.Q THEN
 	_FirstCycle[3]:=FALSE;
	_FirstCycle[4]:=FALSE;
END_IF

{region '新建电动夹爪功能块稳定性测试'}
//CASE  itestStep  OF
//0://等待启动
//		 IF   xtestbutton  THEN
//					ERG_20C_1.stDeviceOpe.xInitControl:=TRUE;
//					ERG_20C_2.stDeviceOpe.xInitControl:=TRUE;
//		 END_IF
//		 IF   ERG_20C_1.stDevice.xQBusy  AND
//				  ERG_20C_2.stDevice.xQBusy	THEN
//					 itestStep:=itestStep +1;
//		 END_IF
//1://等待初始化完成
//		IF  ERG_20C_1.stDevice.xQDone  AND
//				ERG_20C_2.stDevice.xQDone THEN
//					 itestStep:=itestStep +1; 
//		 END_IF
//2://夹爪松开
//	 	 ERG_20C_1.stDeviceOpe.aHMIReleaseButton[1]:=TRUE;
//		 ERG_20C_2 .stDeviceOpe.aHMIReleaseButton[1]:=TRUE;		
//		 IF  	ERG_20C_1.stDevice.xQBusy  AND 
//					ERG_20C_2 .stDevice.xQBusy THEN
//					 itestStep:=itestStep +1;
//		 END_IF
//3://等待夹爪松开完成
//	 	 IF   ERG_20C_1.stDevice.xQDone AND 
//					ERG_20C_2.stDevice.xQDone THEN
//					 itestStep:=itestStep +1;
//		 END_IF
//4://夹爪夹紧
//	 	 ERG_20C_1.stDeviceOpe.aHMIClampButton[1]:=TRUE;
//		 ERG_20C_2.stDeviceOpe.aHMIClampButton[1]:=TRUE;		
//		 IF   ERG_20C_1.stDevice.xQBusy AND 
//					ERG_20C_2.stDevice.xQBusy  THEN
//					 itestStep:=itestStep +1;
//		 END_IF
//5://等待夹爪夹紧完成
//	 	 IF   ERG_20C_1.stDevice.xQDone AND 
//					ERG_20C_2.stDevice.xQDone  THEN
//					 itestStep:=itestStep +1;
//		 END_IF
//6://夹爪旋松
//	 	 ERG_20C_1.stDeviceOpe.aHMIRotateReleaseButton[1]:=TRUE;
//		 ERG_20C_2 .stDeviceOpe.aHMIRotateReleaseButton[1]:=TRUE;
//		 IF   ERG_20C_1.stDevice.xQBusy  AND 
//				  ERG_20C_2.stDevice.xQBusy  THEN
//					 itestStep:=itestStep +1;
//		 END_IF
//7://等待夹爪旋松完成
//	 	 IF   ERG_20C_1.stDevice.xQDone  AND 
//					ERG_20C_2.stDevice.xQDone THEN
//					 itestStep:=itestStep +1;
//		 END_IF
//8://夹爪拧精
//	 	 ERG_20C_1.stDeviceOpe.aHMIRotateClampButton[1]:=TRUE;
//		 ERG_20C_2.stDeviceOpe.aHMIRotateClampButton[1]:=TRUE;		
//		 IF   ERG_20C_1.stDevice.xQBusy AND 
//          ERG_20C_2.stDevice.xQBusy  THEN
//					 itestStep:=itestStep +1;
//		 END_IF
//9://夹爪拧紧
//	 	 IF   ERG_20C_1.stDevice.xQDone AND 
//					ERG_20C_2.stDevice.xQDone THEN
//					 itestStep:=2;
//		 END_IF
//	 		
//END_CASE
END_ACTION

ACTION ILC:

//---------------------------------------------------工站可执行-------------------------------------------------------
station.xCanRun := TRUE ;

//---------------------------------------------------气缸动作条件-------------------------------------------
fbVTCPressCyl_1.xOffILC	:=	TRUE	;
fbVTCPressCyl_1.xOnILC	:=	TRUE	;
fbVTCPressCyl_2.xOffILC	:=	TRUE	;
fbVTCPressCyl_2.xOnILC	:=	TRUE	;
fbVTCPressCyl_3.xOffILC	:=	TRUE	;
fbVTCPressCyl_3.xOnILC	:=	TRUE	;
fbVTCPressCyl_4.xOffILC	:=	TRUE	;
fbVTCPressCyl_4.xOnILC	:=	TRUE	;
fbVTCCyl_1.xOffILC	:=	TRUE	;
fbVTCCyl_1.xOnILC	:=	TRUE	;
fbVTCCyl_2.xOffILC	:=	TRUE	;
fbVTCCyl_2.xOnILC	:=	TRUE	;



//---------------------------------------------------伺服动作条件-------------------------------------------
fbXAxisMove.xRunILC 	:= 		
fbXAxisMove.xMoveILC[1]	:= 		
fbXAxisMove.xMoveILC[2] 	:= 		
fbXAxisMove.xMoveILC[3]	:= 		
fbXAxisMove.xMoveILC[4]	:= 		
fbXAxisMove.xMoveILC[5]	:= 
fbXAxisMove.xMoveILC[6]	:= 	fbVTCCyl_1.xHP_Sensor	AND 	fbVTCCyl_2.xHP_Sensor	;
fbYAxisMove.xRunILC 	:= 		
fbYAxisMove.xMoveILC[1]	:= 		
fbYAxisMove.xMoveILC[2]	:= 		
fbYAxisMove.xMoveILC[3]	:= 		
fbYAxisMove.xMoveILC[4]	:= 		
fbYAxisMove.xMoveILC[5]	:= 	fbVTCCyl_1.xHP_Sensor	AND 	fbVTCCyl_2.xHP_Sensor	;
///电动夹爪
fbERG_20_Modbus[1].xDeviceRunning:=
fbERG_20_Modbus[2].xDeviceRunning:=station.xSingleRunning OR station.xRunning OR station.xIniting;

Camera.xIDeviceRunning:=station.xSingleRunning;
END_ACTION

ACTION TipAuto:
//------------------------------------------------AutoTip Cylinder--------------------------------
//station.adwAutoTip[1].00	:=	fbVTCPressCyl_1.xAutoTip	;
//station.adwAutoTip[1].01	:=	fbVTCPressCyl_2.xAutoTip	;
//station.adwAutoTip[1].02	:=	fbVTCPressCyl_3.xAutoTip	;
//station.adwAutoTip[1].03	:=	fbVTCPressCyl_4.xAutoTip	;
station.adwAutoTip[1].04	:=	fbVTCCyl_1.xAutoTip	;
station.adwAutoTip[1].05	:=	fbVTCCyl_2.xAutoTip	;

//------------------------------------------------AutoTip Servo--------------------------------
//**************************************
//FOR i:= 1 TO 5 BY 1 DO 
//	IF fbXAxisMove.xMoveAuto[i] THEN
//		fbXAxisMove.iPosNumber := i ;
//	END_IF
//	IF fbYAxisMove.xMoveAuto[i] THEN
//		fbYAxisMove.iPosNumber := i ;
//	END_IF
//END_FOR
//IF fbMachine[1].xAutoMode AND NOT fbMachine[1].xRunning  AND  arTonDelay[9].Q  THEN 
//		IF fbXAxisMove.iPosNumber=1 AND NOT fbXAxisMove.xMoveInPos[1] THEN station.adwAutoTip[1].10:=TRUE; END_IF//轴伺服自动时位置不在位置1	
//		IF fbXAxisMove.iPosNumber=2 AND NOT fbXAxisMove.xMoveInPos[2] THEN station.adwAutoTip[1].11:=TRUE; END_IF//轴伺服自动时位置不在位置2	
//		IF fbXAxisMove.iPosNumber=3 AND NOT fbXAxisMove.xMoveInPos[3] THEN station.adwAutoTip[1].12:=TRUE; END_IF//轴伺服自动时位置不在位置3	
//		IF fbXAxisMove.iPosNumber=4 AND NOT fbXAxisMove.xMoveInPos[4] THEN station.adwAutoTip[1].13:=TRUE; END_IF//轴伺服自动时位置不在位置4	
//		IF fbXAxisMove.iPosNumber=5 AND NOT fbXAxisMove.xMoveInPos[5] THEN station.adwAutoTip[1].14:=TRUE; END_IF//轴伺服自动时位置不在位置5	
//END_IF
//IF fbMachine[1].xAutoMode AND NOT fbMachine[1].xRunning  AND  arTonDelay[10].Q  THEN 		
//		
//		IF fbYAxisMove.iPosNumber=1 AND NOT fbYAxisMove.xMoveInPos[1] THEN station.adwAutoTip[1].15:=TRUE; END_IF//轴伺服自动时位置不在位置1	
//		IF fbYAxisMove.iPosNumber=2 AND NOT fbYAxisMove.xMoveInPos[2] THEN station.adwAutoTip[1].16:=TRUE; END_IF//轴伺服自动时位置不在位置2	
//		IF fbYAxisMove.iPosNumber=3 AND NOT fbYAxisMove.xMoveInPos[3] THEN station.adwAutoTip[1].17:=TRUE; END_IF//轴伺服自动时位置不在位置3	
//		IF fbYAxisMove.iPosNumber=4 AND NOT fbYAxisMove.xMoveInPos[4] THEN station.adwAutoTip[1].18:=TRUE; END_IF//轴伺服自动时位置不在位置4	
//		IF fbYAxisMove.iPosNumber=5 AND NOT fbYAxisMove.xMoveInPos[5] THEN station.adwAutoTip[1].19:=TRUE; END_IF//轴伺服自动时位置不在位置5	
//END_IF
//
END_ACTION

ACTION TipManual:
//--------------------------------------------ManualTip------------------------------------------------------

//-------------------------------------------气缸提示---------------------------------------------------------


//-------------------------------------------伺服提示--------------------------------------------------

/////////////////////////////////////////////////////////////////////////////////////////////////////////////////
END_ACTION

ACTION Z_Output:
(**************************气缸输出********************************)
QxS01VTCPressCyl_1WP	:=FALSE;//(NOT  fbMachine[1].xAutoMode AND NOT station.xSingleRunning  AND    fbVTCPressCyl_1.xWP_Valve	) OR
											 			//( (fbMachine[1].xAutoMode OR  station.xsingleRunning ) AND  	fbFlowLine.arQVTCCylWPValve[1]);
QxS01VTCPressCyl_1HP	:=	(NOT  fbMachine[1].xAutoMode AND NOT station.xSingleRunning  AND    fbVTCPressCyl_1.xHP_Valve	) OR
												 ( (fbMachine[1].xAutoMode OR  station.xsingleRunning ) AND  	fbFlowLine.arQVTCCylHPValve[1]);
QxS01VTCPressCyl_2WP	:=FALSE;//	(NOT  fbMachine[1].xAutoMode AND NOT station.xSingleRunning  AND    fbVTCPressCyl_2.xWP_Valve	) OR
															// ( (fbMachine[1].xAutoMode OR  station.xsingleRunning ) AND  	fbFlowLine.arQVTCCylWPValve[2]);
QxS01VTCPressCyl_2HP	:=	(NOT  fbMachine[1].xAutoMode AND NOT station.xSingleRunning  AND    fbVTCPressCyl_2.xHP_Valve	) OR
												 ( (fbMachine[1].xAutoMode OR  station.xsingleRunning ) AND  	fbFlowLine.arQVTCCylHPValve[2]);
QxS01VTCPressCyl_3WP	:=FALSE;//		(NOT  fbMachine[1].xAutoMode AND NOT station.xSingleRunning  AND    fbVTCPressCyl_3.xWP_Valve	) OR
												//	( (fbMachine[1].xAutoMode OR  station.xsingleRunning ) AND  	fbFlowLine.arQVTCCylWPValve[3]);
QxS01VTCPressCyl_3HP	:=	(NOT  fbMachine[1].xAutoMode AND NOT station.xSingleRunning  AND    fbVTCPressCyl_3.xHP_Valve	) OR
												 ( (fbMachine[1].xAutoMode OR  station.xsingleRunning ) AND  	fbFlowLine.arQVTCCylHPValve[3]);
QxS01VTCPressCyl_4WP	:=FALSE;//			(NOT  fbMachine[1].xAutoMode AND NOT station.xSingleRunning  AND    fbVTCPressCyl_4.xWP_Valve	) OR
												//( (fbMachine[1].xAutoMode OR  station.xsingleRunning ) AND  	fbFlowLine.arQVTCCylWPValve[4]);
QxS01VTCPressCyl_4HP	:=		(NOT  fbMachine[1].xAutoMode AND NOT station.xSingleRunning  AND    fbVTCPressCyl_4.xHP_Valve	) OR
												 ( (fbMachine[1].xAutoMode OR  station.xsingleRunning ) AND  	fbFlowLine.arQVTCCylHPValve[4]);
QxS01VTCCyl_1WP	:=	fbVTCCyl_1.xWP_Valve	;
QxS01VTCCyl_1HP	:=	fbVTCCyl_1.xHP_Valve	;
QxS01VTCCyl_2WP	:=	fbVTCCyl_2.xWP_Valve	;
QxS01VTCCyl_2HP	:=	fbVTCCyl_2.xHP_Valve	;
END_ACTION

END_PROGRAM

// ---- POUs/003_FB/05_StationFB/FB_Station.TcPOU
FUNCTION_BLOCK FB_Station
VAR_INPUT
	xEStop						: BOOL;					//急停
	xKey						: BOOL:=TRUE;			//钥匙开关
	xSafety						: BOOL;					//安全防护
	xManualMode					: BOOL;					//手动模式
	xReset						: BOOL;					//复位按钮	
	xMachinePause				: BOOL;					//整机暂停按钮
	xMachineReInit				: BOOL;					//整机重新初始化时，复位初始化完成
	xMachineIniting				: BOOL;					//整机初始化中
	xMachineRunning				: BOOL;					//整机自动中
	tInitTimeout				: TIME:=T#90S;			//初始化超时
	xPauseDisable        		: BOOL;            		//暂停失效标志位
	
	xEmptying					:BOOL;					//工站清空中
	xEmptyDone					:BOOL;					//工站清空结束
	
	
	
	
	xInitHmi					: BOOL;					//初始化HMI
	xInitDone					: BOOL;					//初始化完成
	xDisabled					: BOOL;					//工站屏蔽
	xCycleRunHmi				: BOOL;					//连动HMI
	xJogRunHmi					: BOOL;					//寸动HMI
	xPauseHmi					: BOOL;					//暂停HMI
	xStop						: BOOL;					//其它条件要求工站停止运行
	xSingleRunFlag				: BOOL;					//单动标志
	xCycleEnable				: BOOL;					//循环开始，工站周期计时开始
	rWaitingTime				: REAL;					//周期等待时间，如待料，单位s  
	
	adwAlarm	          		: ARRAY[1..4] OF DWORD;	//报警
	adwAutoTip					: ARRAY[1..4] OF DWORD;	//自动提示
	adwManualTip				: ARRAY[1..4] OF DWORD;	//手动提示
	xAlarm						: BOOL;					//报警中
	xAutoTip					: BOOL;					//自动提示中
	xManualTip					: BOOL;					//手动提示中
	xTip						: BOOL;					//提示中
	xDone						: BOOL;					//工站完成
	xCanRun						: BOOL;					//工站可动作
	iStepAuto           		: INT ;         		//自动流程步
	iStepInit           		: INT ;         		//初始化流程步
	bAutoState					: BYTE ;				//工站自动流程状态机 
	xRunningOffProhibit			: BOOL;					///流程中禁止停止
	xSingleContinuousRun		: BOOL;					///连续测试运行
END_VAR

VAR_OUTPUT
	xStationIniting				: BOOL;					//单工站初始化中
	xIniting					: BOOL;					//初始化中
	xInitTimeout				: BOOL;					//初始化超时
	xCycleRunning				: BOOL;					//连动中
	xJogRunning					: BOOL;					//寸动中
	xSingleRunning				: BOOL;					//单动中
	xRunning					: BOOL;					//运行中
	xDeviceRunning		: BOOL;					//第三方设备运行中
	uiState						: UINT;					//工站状态
	//tCycleTime				:TIME;
	diCycleTime 				: DINT;					//基础时间是100ms
	diLastCycleTime				: DINT;					//基础时间是100ms
	QstrStepInitDescription		: STRING[50];			//初始化描述
	QstrStepAutoDecription		:STRING[50];			//自动步骤描述
	xQStepAutoTrans				:BOOL;					//自动步跳转
	xQStepInitTrans				:BOOL;					//初始化步跳转
	
	xQSingleContinuousRunning		: BOOL;					///连续测试运行中
END_VAR

VAR
	{attribute 'hide'}
	ftInitHmi					: F_TRIG;				//初始化HMI上升沿
	{attribute 'hide'}
	rtMachineReInit				: R_TRIG;				//整机重新初始化上升沿
	{attribute 'hide'}
	xInitAble					: BOOL;					//初始化条件
	{attribute 'hide'}
	xRunAble					: BOOL;					//运行条件
	{attribute 'hide'}
	tonInitTimeout				: TON;					//初始化超时计时
	{attribute 'hide'}
	ftCycleRunHMI				: F_TRIG;				//连动HMI上升沿
	{attribute 'hide'}
	rtJogRunHMI					: R_TRIG;				//寸动HMI上升沿
	{attribute 'hide'}
	xPause						: BOOL;					//暂停
	{attribute 'hide'}
	lrCycleTimer					: LREAL;				//计时器，单位100ns，除于10000后单位ms
	{attribute 'hide'}
	lrWaitingTimer				: LREAL;				//等待时间计时器
	{attribute 'hide'}
	rtCycleTimeStop				: R_TRIG;				//工站周期计时停止上升沿
	
	ton_AutoTimeout				:TON;					//工站自动流程超时			//自动程序有BUG
	i : INT ;
	xFirstCycle : BOOL ;	
	{attribute 'hide'}
	rStationStart	  : R_TRIG;							//工站完成上升沿
	{attribute 'hide'}
	fStationRunning : R_TRIG;
	{attribute 'hide'}
	iOldStepAuto           		: INT ;         		//自动流程步历史
	{attribute 'hide'}
	iOldStepInit           		: INT ;         		//初始化流程历史
	{attribute 'hide'}
	OldStepAutoR_TRIG						:R_TRIG;
	{attribute 'hide'}
	OldStepInitR_TRIG						:R_TRIG;
END_VAR

ACT_General();
ACT_Init();
ACT_Run();
ACT_State();
ACT_CycleTime();
ACT_Logfile();

ACTION ACT_CycleTime:
//	初始化时同时初始化工站周期计时
IF xIniting THEN
	xCycleEnable:=FALSE;
END_IF

//工站完成触发信号
rStationStart(CLK:= xCycleEnable);
IF rStationStart.Q 
THEN
	diCycleTime:=diLastCycleTime;
	diLastCycleTime := 0;
END_IF
//	工站周期计时
IF xRunning AND xCycleEnable AND stSysPulse.xR100ms
THEN
	diLastCycleTime := diLastCycleTime + 1;//对应最小周期是0.1ms
END_IF
END_ACTION

ACTION ACT_General:
//	报警中
FOR i:=1 TO 4 BY 1 DO 
		  xAlarm := FALSE ;
	 IF adwAlarm[i]<>0 THEN 
		  xAlarm := TRUE ;
			EXIT ;
	 END_IF
END_FOR

//	提示中
FOR i:=1 TO 4 BY 1 DO 
		  xAutoTip := FALSE ;
	 IF adwAutoTip[i]<>0 THEN 
		  xAutoTip := TRUE ;
			EXIT ;
	 END_IF
END_FOR
FOR i:=1 TO 4 BY 1 DO 
		  xManualTip := FALSE ;
	 IF adwManualTip[i]<>0 THEN 
		  xManualTip := TRUE ;
			EXIT ;
	 END_IF
END_FOR
xTip:=xAutoTip
	OR xManualTip;

//	暂停
xPause:=xMachinePause
	OR xPauseHmi
	OR xStop;

//	报警复位
IF xReset THEN
	FOR i:=1 TO 4 BY 1 DO 
		adwAutoTip[i] := adwAlarm[i] := adwManualTip[i] := 0;
	END_FOR
END_IF
END_ACTION

ACTION ACT_Init:
//	初始化条件
xInitAble:=xEStop
	AND xKey
	AND xSafety
	AND xManualMode
	AND NOT xAlarm
	AND NOT xInitTimeout;

//	急停或初始化时先复位初始化完成
ftInitHmi(CLK:=xInitHmi, Q=>);
rtMachineReInit(CLK:=xMachineReInit, Q=>);

IF ((NOT xEStop OR rtMachineReInit.Q OR ftInitHmi.Q )AND gc_xEstopYesORno)OR 
	 (( rtMachineReInit.Q OR ftInitHmi.Q AND xInitAble)AND NOT gc_xEstopYesORno)
THEN
	xInitDone:=FALSE;
END_IF

//	单工站初始化中
IF xInitAble
	AND NOT xInitDone
	AND NOT xInitTimeout
	AND NOT xPause
	AND NOT xMachineIniting
THEN
	IF ftInitHmi.Q THEN
		xStationIniting:=TRUE;
	END_IF
ELSE
	xStationIniting:=FALSE;
END_IF

//	初始化中
xIniting:=xStationIniting
	OR xMachineIniting
		AND xInitAble
		AND NOT xInitDone;

//	初始化超时
tonInitTimeout(
	IN:=xIniting,
	PT:=tInitTimeout,
	Q=>, ET=>);
IF xReset THEN
	xInitTimeout:=FALSE;
END_IF
IF tonInitTimeout.Q THEN
	xInitTimeout:=TRUE;
END_IF
END_ACTION

ACTION ACT_Logfile:
//********************************//
IF iOldStepAuto=iStepAuto THEN
	xQStepAutoTrans:=FALSE;
END_IF
IF    iOldStepAuto<>iStepAuto THEN
	xQStepAutoTrans:=TRUE;
	iOldStepAuto:=iStepAuto;
END_IF

IF  iOldStepInit=iStepInit THEN
	xQStepInitTrans:=FALSE;
END_IF

IF    iOldStepInit<>iStepInit THEN
	xQStepInitTrans:=TRUE;
	iOldStepInit:=iStepInit;
END_IF
END_ACTION

ACTION ACT_Run:
//	运行条件
xRunAble:=xEStop
	AND xKey
	AND xSafety
	AND xInitDone
	AND NOT xAlarm
	AND NOT xAutoTip;

//	单动标志
ftCycleRunHMI(CLK:=xCycleRunHmi, Q=>);
rtJogRunHmi(CLK:=xJogRunHmi, Q=>);
IF xEStop
	AND xInitDone
THEN
	IF (ftCycleRunHMI.Q
			OR rtJogRunHmi.Q)
		AND xRunAble
		AND xManualMode
	THEN
		xSingleRunFlag:=TRUE;
	END_IF
ELSE
	xSingleRunFlag:=FALSE;
END_IF

//	连动中、寸动中
IF xRunAble
	AND xManualMode
	AND xSingleRunFlag
	AND NOT xPause
THEN
	IF ftCycleRunHMI.Q THEN
		xCycleRunning:=TRUE;
	END_IF
	xJogRunning:=rtJogRunHmi.CLK;
ELSE
	xCycleRunning:=FALSE;
	xJogRunning:=FALSE;
END_IF

//	单动中
xSingleRunning:=xCycleRunning
	OR xJogRunning;

//	运行中
xRunning:=xSingleRunning
	OR xMachineRunning
		AND xRunAble;

xDeviceRunning := xRunning OR xIniting;		
		
//工站自动流程超时

//ton_AutoTimeout(IN:= bRunning 
//					AND NOT bSingleRunFlag 
//					AND bCycleStart , PT:=T#35S , Q=> , ET=> );		//自动程序有BUG

(**********************连续单循环标志位************************)
IF  xSingleContinuousRun THEN
		xQSingleContinuousRunning:=true;
else
		xQSingleContinuousRunning:=FALSE;
END_IF
END_ACTION

ACTION ACT_State:


//	未准备好
IF NOT xInitDone
	AND NOT xAlarm
THEN
	uiState:=E_State.NotReady;
END_IF

//	运行中
IF xRunning THEN
	uiState:=E_State.iRunning;
END_IF

//	报警中
IF xAlarm THEN
	uiState:=E_State.Alarm;
END_IF

//	准备好
IF xInitDone
	AND NOT xAlarm
	AND NOT xRunning
THEN
	uiState:=E_State.Ready;
END_IF

//工站完成
IF xInitDone AND xDone THEN 
	uiState:=E_State.Done;
END_IF
END_ACTION

END_FUNCTION_BLOCK

// ---- POUs/003_FB/10_CylinderFB/FB_Cylinder.TcPOU
FUNCTION_BLOCK FB_Cylinder
VAR_INPUT
	xEStop						: BOOL;					//急停
	xSafety						: BOOL;					//安全防护
	xManualMode					: BOOL;					//手动模式
	xAutoMode					: BOOL;					//自动模式
	xAirOn						: BOOL;					//气压正常
	tAlarm						: TIME:=T#5S;			//报警延时
	xReset					: BOOL;					//报警复位,提示复位
	xAlarmDisable               : BOOL;                 //报警屏蔽
	
	xHmi						: BOOL;					//手动HMI
	xManual						: BOOL;					//手动执行
	xAuto						: BOOL;					//自动执行
	xInit						: BOOL;					//初始化执行
	xRelease					: BOOL;					//输出释放，气缸泄气
	xOnILC						: BOOL;			        //动作条件
	xOffILC						: BOOL;			        //复位条件
	xHP_Sensor					: BOOL;					//原点感应器
	xWP_Sensor					: BOOL;					//动点感应器
	tHP_Delay					: TIME;					//原点延时
	tWP_Delay					: TIME;					//动点延时
	byManualTip					: BYTE;					//手动提示字节，多个提示，用于外部触发
	xManualTip					: BOOL;					//手动提示，单个提示，用于外部触发
	xTryRun						:BOOL;					//空运行
END_VAR

VAR_OUTPUT
	xHP_Valve					: BOOL;					//原点阀
	xWP_Valve					: BOOL;					//动点阀
	xHP_Delay					: BOOL;					//原点状态
	xWP_Delay					: BOOL;					//动点状态
	xHP_Off						: BOOL;					//原点无信号
	xWP_Off						: BOOL;					//动点无信号
	xHP_On						: BOOL;					//原点应为Off
	xWP_On						: BOOL;					//动点应为Off
	xAutoTip					: BOOL;					//自动提示，用于外部触发
	xAlarming					: BOOL;					//报警中
	xBusy						: BOOL;					//运动中
END_VAR

VAR
	{attribute 'hide'}
	ftHmi						: F_TRIG;				//手动HMI下降沿
	{attribute 'hide'}
	rtManual					: R_TRIG;				//手动执行上升沿
//	{attribute 'hide'}
	xEnable						: BOOL;					//使能
	{attribute 'hide'}
	tonHP_Delay					: TON;					//原点延时计时
	{attribute 'hide'}
	tonWP_Delay					: TON;					//动点延时计时
	{attribute 'hide'}
	tAlarmTime					: TIME;					//报警延时
	{attribute 'hide'}
	tonHP						: TON;					//原点输出计时
	{attribute 'hide'}
	tonWP						: TON;					//动点输出计时
END_VAR

ACT_Manual();
ACT_Output();
ACT_Delay();
ACT_Alarm();
ACT_Tip();

ACTION ACT_Alarm:
//	延时设置，防止报警延时小于到位延时误报警
IF tAlarm > MAX(tHP_Delay, tWP_Delay) THEN
	tAlarmTime:=tAlarm;
ELSE
	tAlarmTime:=tAlarm + MAX(tHP_Delay, tWP_Delay);
END_IF

//	报警延时
tonHP(IN:=xAirOn AND xHP_Valve, PT:=tAlarmTime, Q=>, ET=>);
tonWP(IN:=xAirOn AND xWP_Valve, PT:=tAlarmTime, Q=>, ET=>);

//	先报警复位
IF xReset THEN
	 xHP_Off:=FALSE;
	 xWP_Off:=FALSE;
	 xHP_On:=FALSE;
	 xWP_On:=FALSE;
END_IF

//	报警输出，Off报警用延时，On报警用感应器，防止感应器抖动时无到位无报警
IF tonHP.Q AND NOT xAlarmDisable THEN
	IF NOT xHP_Delay THEN
		xHP_Off:=TRUE;
	END_IF
	IF xWP_Sensor THEN
		xWP_On:=TRUE;
	END_IF
END_IF
IF tonWP.Q AND NOT xAlarmDisable THEN
	IF NOT xWP_Delay THEN
		xWP_Off:=TRUE;
	END_IF
	IF xHP_Sensor THEN
		xHP_On:=TRUE;
	END_IF
END_IF

xAlarming:=(xHP_Off OR xWP_Off OR xHP_On OR xWP_On) AND NOT xAlarmDisable;

xBusy:=NOT xAlarming
	AND (xHP_Valve AND NOT xHP_Delay
		OR xWP_Valve AND NOT xWP_Delay);
END_ACTION

ACTION ACT_Delay:
//	原点延时
tonHP_Delay(
	IN:=xHP_Valve
		AND NOT xWP_Valve
		AND xHP_Sensor 
		AND NOT xWP_Sensor,
	PT:=tHP_Delay,
	Q=>xHP_Delay,
	ET=>);

//	动点延时
tonWP_Delay(
	IN:=NOT xHP_Valve
		AND xWP_Valve
		AND NOT xHP_Sensor
		AND (xWP_Sensor OR xTryRun),
	PT:=tWP_Delay,
	Q=>xWP_Delay,
	ET=>);
END_ACTION

ACTION ACT_Manual:
//	手动操作
ftHmi(CLK:=xHmi, Q=>);
IF ftHmi.Q
	AND xEStop
	AND xSafety
	AND xManualMode
	AND xAirOn
	AND ((
			xManual = xAuto
			AND xOnILC
		)
		OR (
			(xManual XOR xAuto)
			AND xOffILC
		)
	)
THEN
	xManual:=NOT xManual;
END_IF

//	初始化时复位手动执行//复位自动执行
IF xInit THEN
	xManual:=FALSE;
	xAuto  :=FALSE;
END_IF
END_ACTION

ACTION ACT_Output:
//	使能
rtManual(CLK:=xManual, Q=> );
IF xEStop THEN
	IF rtManual.Q
		OR xInit
	THEN
		xEnable:=TRUE;
	END_IF
ELSE
	;//xEnable:=FALSE;
END_IF

//	原点阀输出
xHP_Valve:=xEnable
	AND NOT xRelease
	AND (xManual = xAuto);

//	动点阀输出
xWP_Valve:=xEnable
	AND NOT xRelease
	AND (xManual XOR xAuto);
	
//	自动复位
xInit:=FALSE;
//xHmi:=FALSE;
END_ACTION

ACTION ACT_Tip:
IF xReset THEN
	xManualTip:=FALSE;
	byManualTip:=0;
END_IF

xAutoTip:=xAutoMode AND xManual;
END_ACTION

END_FUNCTION_BLOCK

// ---- POUs/003_FB/0004_FlowLine/FB_FlowLine.TcPOU
FUNCTION_BLOCK FB_FlowLine
(*
********************************************************************************
* Name: FB_Camera
*
* Author:  AutomanH
* Version: 1.0.0
*
* Description:
*	Flow Line Program and motor control
*
* Remarks:
*
*
* Revisions:
*   V1.0.0 -Automanh 2022.06.08
* 	V1.1.0-Automanh 2022.06.20,Add ACT_Motor();
*		V2.0.0-Automanh 2022.07.18 add timeout alarm 
*********************************************************************************)
VAR_INPUT
 arIReachedSensor:ARRAY[1..iColumnsNum] OF BOOL;
 arIVTCCylHPSensor:ARRAY[1..iColumnsNum] OF BOOL;
 arIVTCCylWPSensor:ARRAY[1..iColumnsNum] OF BOOL;
 xIRunningPremit:BOOL;
 xIMotorStop:BOOL;
 xIEmptyDone:BOOL;
 xITryRun:BOOL;
 xIMotorEstop:BOOL;
 xIInit:BOOL;
 xIMotorStartButtonHmi:BOOL;
 xIMotorStopButtonHmi:BOOL;
 xIManualMode:BOOL;
 xIAutoMode:BOOL;
 xIDeviceRunning:BOOL;
END_VAR
VAR_OUTPUT
 arQVTCCylHPValve:ARRAY[1..iColumnsNum] OF BOOL;
 arQVTCCylWPValve:ARRAY[1..iColumnsNum] OF BOOL; 
 xQMotorEstop:BOOL;
 xQMotorStop:BOOL;
 xQMotorStart:BOOL;
 xQBusy:BOOL;
 xQError:BOOL;
 xQDone:BOOL;
END_VAR
VAR
 	//链板线电机启动
 	xMotorStart:BOOL;
	xMotorStop:BOOL;
	// 链板线步骤
	bFlowLineStep: BYTE;
	bFlowLineStepOld:BYTE;
	bMotorCtrlStep:BYTE;
	// 延时
	arTonDelay: ARRAY[1..10] OF Tc2_Standard.TON;
	i:INT;
	_xFirstCycle: BOOL;
	stMotorStatus:DUT_Motor;
	ModeSwitchR_TRIG:R_TRIG;
	MotorStopR_TRIG:R_TRIG;
	InitR_TRIG:R_TRIG;
	bInitStep: BYTE;
	//超时
	tTimeOut:TON;
	
END_VAR
VAR CONSTANT
 	iColumnsNum :INT:=4;
END_VAR

ACT_Motor();
ACT_Flow();
ACT_Manual();
ACT_Init();

ACTION ACT_Flow:


{region "链板线程序"}
tTimeOut(IN:= bFlowLineStepOld =bFlowLineStep AND bFlowLineStepOld<>0,PT:=T#15S , Q=> , ET=> );
IF  tTimeOut.Q THEN
		xQError:=TRUE; 
		tTimeOut(IN:=FALSE); 			
END_IF
	CASE bFlowLineStep OF
	0://启动
		FOR i:=1 TO 10 BY 1 DO
			arTonDelay[i](IN:=FALSE);
		END_FOR
		IF	xIRunningPremit  AND NOT xIEmptyDone  THEN
				bInitStep:=0;
				xMotorStart:=TRUE;
				xMotorStop:=FALSE;
				_xFirstCycle:=TRUE;
				xIRunningPremit:=FALSE;
				xQBusy:=TRUE;
				xQDone:=FALSE;
				bFlowLineStep:=bFlowLineStep +1;
		ELSE
				xMotorStart:=FALSE;
		END_IF
	1://下压气缸回原
		 		bFlowLineStepOld :=bFlowLineStep;
				FOR  i:=1 TO iColumnsNum BY 1 DO
					 arQVTCCylWPValve[i]:=FALSE;
					 arQVTCCylHPValve[i]:=TRUE;
				END_FOR 	
				bFlowLineStep:=bFlowLineStep +1;
	2://判断回原是否完成
		 	bFlowLineStepOld :=bFlowLineStep;
				FOR  i:=1 TO iColumnsNum BY 1 DO
					IF  NOT arIVTCCylHPSensor[i] THEN
						EXIT;	
					 ELSIF  i  =iColumnsNum THEN
							bFlowLineStep:=bFlowLineStep +1;
					 END_IF
				 END_FOR
	3://到位传感器检测
		// bFlowLineStepOld :=bFlowLineStep;
		IF NOT xITryRun THEN
			FOR  i:=1 TO iColumnsNum BY 1 DO
				IF  NOT arIReachedSensor[i]  THEN
					EXIT;
				ELSIF   i =iColumnsNum THEN
					bFlowLineStep:=bFlowLineStep +1;
				END_IF
			END_FOR
		ELSE
				bFlowLineStep:=bFlowLineStep +2;
		END_IF
	4://下压气缸伸出
		 			bFlowLineStepOld :=bFlowLineStep;
					FOR  i:=1 TO iColumnsNum BY 1 DO
							 arQVTCCylWPValve[i]:=TRUE;
							 arQVTCCylHPValve[i]:=FALSE;
					 
					END_FOR
						bFlowLineStep:=bFlowLineStep +1;
	5://检测下压气缸到位
		 		bFlowLineStepOld :=bFlowLineStep;
				bFlowLineStep:=bFlowLineStep +1;
	6://延时1s
		 	bFlowLineStepOld :=bFlowLineStep;
			arTonDelay[3](IN:=TRUE  , PT:=T#1S , Q=> , ET=> );
			IF  	arTonDelay[3].Q THEN
						bFlowLineStep:=bFlowLineStep +1;
						arTonDelay[3](IN:=FALSE);
			END_IF	      
	7://输出链板线Ready信号
		 	bFlowLineStepOld :=bFlowLineStep;
			 xQBusy:=FALSE;
			 xQDone:=TRUE;
			 bFlowLineStep:=0;
	END_CASE
	xIRunningPremit:=FALSE;
{endregion}
END_ACTION

ACTION ACT_Init:
InitR_TRIG(CLK:= xIInit, Q=> );
CASE bInitStep OF
 0:
		IF	InitR_TRIG.Q THEN
				bFlowLineStep:=0;
				xQBusy:=FALSE;
				xQError:=FALSE;
				bFlowLineStepOld:=0;
				bInitStep:=bInitStep +1;
		 END_IF
 1://气缸回原
			FOR  i:=1 TO iColumnsNum BY 1 DO
			 	 arQVTCCylWPValve[i]:=FALSE;
				 arQVTCCylHPValve[i]:=TRUE;
			END_FOR 	
				bInitStep:=bInitStep +1;
 2://链板线停止
 			xQMotorEstop:=FALSE;
		  xQMotorStop:=FALSE;
		  xQMotorStart:=FALSE;
			xQBusy:=FALSE;
			bInitStep:=0;
END_CASE
xIInit:=FALSE;
END_ACTION

ACTION ACT_Manual:
IF  (xMotorStart AND  xIDeviceRunning )  OR
 		(xIMotorStartButtonHmi AND xIManualMode) THEN
				xMotorStart:=TRUE;
				xMotorStop:=FALSE;
ELSIF
 	 (xIMotorStop AND  xIDeviceRunning )  OR
 	(xIMotorStopButtonHmi AND xIManualMode)	THEN
			xMotorStart:=FALSE;
			xMotorStop:=TRUE;
END_IF
END_ACTION

ACTION ACT_Motor:
ModeSwitchR_TRIG(CLK:= xIManualMode (*XOR xIAutoMode*) , Q=> );
CASE  bMotorCtrlStep  OF
0://等待激活
			IF   xIMotorEstop THEN
			 		bMotorCtrlStep:=1;
			ELSIF xMotorStop	 THEN
			 		bMotorCtrlStep:=2;
			ELSIF ModeSwitchR_TRIG.Q THEN
			 		bMotorCtrlStep:=4;
			ELSIF xMotorStart	 THEN
			 		bMotorCtrlStep:=3;
			END_IF
1://急停被拍下
		xQMotorEstop:=TRUE;
		xQMotorStart:=FALSE;
		bMotorCtrlStep:=0;
2://停止被按下
		xQMotorStart:=FALSE;
		xQMotorStop:=TRUE;
		bMotorCtrlStep:=0;
3://启动被按下
			xQMotorStop:=FALSE;
			xQMotorStart:=TRUE;
			bMotorCtrlStep:=0;
4://设备模式切换
			xQMotorStart:=FALSE;
			xQMotorStop:=TRUE;
			bMotorCtrlStep:=0;
			bFlowLineStep:=0;
END_CASE
END_ACTION

END_FUNCTION_BLOCK

// ---- POUs/003_FB/19-AxisFB/FB_Axis.TcPOU
FUNCTION_BLOCK FB_Axis
VAR_INPUT
	xEStop								: BOOL;					//急停
	xKey									: BOOL;					//钥匙开关
	xSafety								: BOOL;					//安全防护
	xManualMode						: BOOL;					//手动模式
	xAutoMode							: BOOL;					//自动模式
	xAlarmReset						: BOOL;					//报警复位
	                  		
	xStop									: BOOL;					//轴停止
	xHalt									: BOOL;					//轴暂停
	xSv_not_power					: BOOL;					//轴断使能
	xNotPower       			: BOOL;					//轴断使能
	                  		
	xEnablePositive 			: BOOL:=TRUE;			//允许正转
	xEnableNegative				: BOOL:=TRUE;			//允许反转
	xRunILC								: BOOL:=TRUE;			//运行条件
	
	xPowerHmi							: BOOL;					//使能手动HMI
	xSetPosHmi						: BOOL;					//设置零点手动HMI
	xHomeHmi							: BOOL;					//原点搜索HMI
	xAlarmResetHmi				: BOOL;					//报警复位HMI
	xJogForwardHmi				: BOOL;					//Jog+HMI
	xJogBackwardsHmi			: BOOL;					//Jog-HMI
	xStopHmi					: BOOL;
	xJogForwardLimit  		: BOOL ;//JOG+极限
	xJogBackwardsLimit		: BOOL ;//JOG-极限
	
	xITarMoveHmi				:INT;//触摸屏选择 MMove Position
	xITarMoveButtonHmi			:BOOL;//触摸屏中目标位置按钮
	
	xPowerInit						: BOOL;					//使能初始化执行
	xHomeAuto							: BOOL;					//原点搜索自动执行
	xReferenceAuto				:BOOL;					//原点搜索自动执行(用于AxisHome）
	xReferenceHmi					:BOOL;					//原点搜索自动执行(用于AxisHome）
	xCalibrationCam				: BOOL;					//原点校准
	xJogForwardAuto				: BOOL;					//Jog+自动执行
	xJogBackwardsAuto			: BOOL;					//Jog-自动执行
	
	xSingleRun					:BOOL;					//伺服单循环执行，（环形线就是走固定位置）
	
	nMoveNum							: USINT:=6;				//轴绝对定位数量
	xMoveILC							: ARRAY[1..gc_uiAxisMoveNum] OF BOOL:=[gc_uiAxisMoveNum(TRUE)];//绝对定位动作条件
	xMoveHmi							: ARRAY[1..gc_uiAxisMoveNum] OF BOOL;//绝对定位手动Hmi
	xMoveAuto							: ARRAY[1..gc_uiAxisMoveNum] OF BOOL;//绝对定位自动执行
	
	rJogVelocity					: REAL;					//轴Jog速度
	rManualVelocity				: REAL;				//轴手动速度
	rAutoVelocity					: REAL;					//轴自动速度
	rMovePosition					: ARRAY[1..gc_uiAxisMoveNum] OF REAL;//绝对定位位置
	rMoveVelocity					: ARRAY[1..gc_uiAxisMoveNum] OF REAL;//绝对定位速度
	tInPosition						: ARRAY[1..gc_uiAxisMoveNum] OF TIME;//绝对到位延时
	rJogAcceleration      : REAL;                 //轴Jog加速度
	rJogDeceleration      : REAL;                 //轴Jog减速度
	rMoveAcceleration     : REAL;            //轴定位加速度                   	
	rMoveDeceleration     : REAL;           //轴定位减速度 
	rRelativeDistance			: REAL;					//相对定位位置
	rRelativeVelocity			: REAL;					//相对定位速度	
	rVelocityVel			    : REAL;					//连续运行速度
	rVelocityAcc			    : REAL;					//连续运行加速度
	rVelocityDec			    : REAL;					//连续运行减速度	
	
	iPosNumber						: INT;					//位置保存编号

	xRelativeILC        	: BOOL;                 //Relative条件
	xRelativeHmi			    : BOOL;					//相对定位手动Hmi
	xRelativeAuto			    : BOOL;					//相对定位自动执行
	
	xVelocityILC       		: BOOL;                 //Velocity条件
	xVelocityAuto			    : BOOL;					//连续运行启动
	xVelocityDirection		: BOOL;                 //连续运行方向  

	
	xModulo								: BOOL;					//模长内定位启动
	rModuloPosition				: REAL;					//模长内定位位置
	rModuloVelocity				: REAL;					//模长内定位速度
	nModuloDirection			: INT := (MC_Direction.MC_Positive_Direction);//模长定位方向
	tMoveTimeout					: TIME:=T#360S;			//定位超时
	wManualTip						: BYTE;					//手动提示字节,用于外部触发
	{attribute 'hide'}
	iHomingMode     : INT ; //回原模式输入
	{attribute 'hide'}
	xIsLinearMode : BOOL := TRUE;//默认都是线性模式	
	
	xIRefSwitch: BOOL;
	xIRelative_Encoder:BOOL;
	xIResetRefPosCheck: BOOL;
	lrIRefVeloPlusFast: REAL;
	lrIRefVeloMinusFast: REAL;
	lrIRefVeloPlusSlow: REAL;
	lrIRefVeloMinusSlow: REAL;
	lrIReferencePosition:REAL;
END_VAR

VAR_OUTPUT
	xPowerOn							: BOOL;					//使能On
	xSetPosFinish					: BOOL;					//设置零点完成
	xReady								: BOOL;					//准备好
	xMoveDone							: ARRAY[1..gc_uiAxisMoveNum] OF BOOL;//绝对定位完成
	xMoveInPos						: ARRAY[1..gc_uiAxisMoveNum] OF BOOL;//绝对定位到位
	xMoveTimeout					: BOOL;					//定位超时报警
	xNotPowerOn						: BOOL;					//使能未On提示
	
	xError								: BOOL;					//错误
	xbusy									: BOOL;
	nErrorID							: UDINT;				//错误ID
	nErrorCode						: UDINT;				//错误代码
	
	rSetTorque						: REAL;					//设定转矩
	rSetPos								: REAL;					//设定位置
	rModuloSetPos					: REAL;					//模长内定位设定位置
	rModuloSetTurns				: REAL;					//模长内定位设定匝数
	rTargetPos						: REAL;					//目标位置
	
	rActTorque						: REAL;					//当前转矩
	rActPos								: REAL;					//当前位置
	rActVelo							: REAL;					//当前速度
	rModuloActPos					: REAL;					//模长内定位当前位置
	rModuloActTurns				: REAL;					//模长内定位当前匝数
	rPosDiff							: REAL;					//跟随误差

	xRelativeDone1				: BOOL;					//相对定位完成标志	
	xRelativeDone					: BOOL;					//相对定位完成
	xRelativeBusy					: BOOL;					//相对定位Busy
	xRelativeError				: BOOL;					//相对定位错误
	udiRelativeErrorID		: UDINT;				//相对定位错误ID
	
	xVelocityInVel				: BOOL;					//连续运行速度到达
	xVelocityBusy					: BOOL;					//连续运行Busy
	xVelocityError				: BOOL;					//连续运行错误
	udiVelocityErrorID		: UDINT;				//连续运行错误ID	
	
	
	xQTarPosition			:REAL;//触摸屏中显示在目标位置中
	xQTarVelocity			:REAL;//触摸屏中显示在目标速度中
	{attribute 'hide'}
	NcToPlc								: NCTOPLC_AXIS_REF;		//轴NcToPlc结构体
	{attribute 'hide'}
	Status								: ST_AxisStatus;		//轴状态结构体
	
	lrQReferenceCheckDiff: REAL;
	lrQPositionAct: REAL;
	lrQReferenceEndPos: REAL;
	xQReferenceEndPosOk: BOOL;
	
END_VAR

VAR_IN_OUT
	{attribute 'hide'}
	Axis									: AXIS_REF;				//轴
END_VAR

VAR
	{attribute 'hide'}
	rtPowerHmi						: R_TRIG;				//使能手动HMI上升沿
	{attribute 'hide'}
	rtSetPosHmi						: R_TRIG;				//设置零点手动HMI上升沿
	{attribute 'hide'}
	xPowerManual					: BOOL;					//使能手动执行
	{attribute 'hide'}
	xPowerAuto						: BOOL;					//使能自动执行
	{attribute 'hide'}
	xPowerEnable					: BOOL;					//使能Enable
	{attribute 'hide'}
	rtPowerOn							: R_TRIG;				//使能上升沿
	{attribute 'hide'}
	rtPowerOff						: R_TRIG;				//使能下降沿
	{attribute 'hide'}
	xRunable							: BOOL;					//可运行
	{attribute 'hide'}
	xHomeManual						: BOOL;					//回原点手动执行
	{attribute 'hide'}
	xHomeExecute					: BOOL;					//回原点触发
	{attribute 'hide'}
	xSetPosExecute				: BOOL;					//设置零点触发
	{attribute 'hide'}
	xResetExecute					: BOOL;					//复位
	{attribute 'hide'}
	xJogForwardManual			: BOOL;					//Jog+手动执行
	{attribute 'hide'}
	xJogBackwardsManual		: BOOL;					//Jog-自动执行
	{attribute 'hide'}
	xJogForward						: BOOL;					//Jog+
	{attribute 'hide'}
	xJogBackwards					: BOOL;					//Jog-
	{attribute 'hide'}
	xMoveManual						: ARRAY[1..gc_uiAxisMoveNum] OF BOOL;//绝对定位手动执行
	{attribute 'hide'}
	xMoveExecute					: ARRAY[1..gc_uiAxisMoveNum] OF BOOL;//绝对定位启动使能
	{attribute 'hide'}
	xRelativeExecute			: BOOL;					//相对定位启动
	{attribute 'hide'}
	xModuloExecute				: BOOL;					//模长内定位启动
	{attribute 'hide'}
	xVelocityExecute			: BOOL;					//相对定位启动
	{attribute 'hide'}
	xVelocityAble			    : BOOL;					//相对定位使能
	{attribute 'hide'}
	rVelocity							:	REAL;					//定位速度
	{attribute 'hide'}
	nIndex 								:	INT;//索引
	{attribute 'hide'}
	tonInPosition					: ARRAY[1..gc_uiAxisMoveNum] OF TON;//绝对定位到位计时
	{attribute 'hide'}
	tonMoveTimeout				: ARRAY[1..gc_uiAxisMoveNum] OF TON;//绝对定位超时
	{attribute 'hide'}
	nIndexMove						: INT;					//绝对定位索引
	{attribute 'hide'}
	xHaltExecute					: BOOL;					//轴暂停
	{attribute 'hide'}
	xStopExecute					: BOOL;					//轴停止
	{attribute 'hide'}
	fbReadStatus					: MC_ReadStatus;		//读取状态功能块
	{attribute 'hide'}
	fbPower								: MC_Power;				//使能功能块
	{attribute 'hide'}
	fbJog									: MC_Jog;				//Jog功能块
	{attribute 'hide'}
	fbHome								: MC_Home;				//原点搜索功能块
	{attribute 'hide'}
	fbMove								: ARRAY[1..gc_uiAxisMoveNum] OF MC_MoveAbsolute;//绝对定位功能块
	{attribute 'hide'}
	fbRelative					: MC_MoveRelative;		//相对定位功能块
	{attribute 'hide'}
	fbVelocity						: MC_MoveVelocity;	    //轴速度运行功能块
	{attribute 'hide'}
	fbModulo							: MC_MoveModulo;		//模长内定位
	{attribute 'hide'}
	fbReset								: MC_Reset;				//错误复位功能块
	{attribute 'hide'}
	fbHalt								: MC_Halt;				//轴暂停功能块
	{attribute 'hide'}
	fbStop								: MC_Stop;				//轴停止功能块
	{attribute 'hide'}
	fbSetPos							: MC_SetPosition;		//设置原点位置

	
	xTarMoveExecute							: ARRAY[1..gc_uiAxisMoveNum] OF BOOL;
	wActionHomeStep:WORD;
	fbReferenceWait: TON;
	fbReferenceEndWait: TON;
	
	tHomeR_TRIG:R_TRIG;
	{attribute 'hide'}
	fbAdsRead			: ADSREAD;
	{attribute 'hide'}
	fbAdsWrite			: ADSWRITE;
	{attribute 'hide'}
	uiencoderId			:UDINT;
	wActionStep				:WORD;
	{attribute 'hide'}
	tAxisCalibR_TRIG		:R_TRIG;
	rReferencePositionoffset		:LREAL	:=0.0;
	xPoweroff	:BOOL;
	
	
	tHomeTimeOut: Ton;
	_RunOverHomeSensorflag: BOOL;
END_VAR

VAR CONSTANT
	NCIDXG_AXPARMS			: UDINT := 16#00004000;	(* Axis with ID: Parameter 			*);
	NCIDXG_ENCPAMS			:UDINT:=16#00005000;	(* Encoder with ID: Parameter 			*);
	uiOffsetEncoderId			:UDINT	:= 16#00010001;	(* Encoder-ID *)
	uiLenEncoderId				:UDINT	:= 4;
	uiPositionBias				:UDINT	:= 16#00000007;	(* Reference position offset*)
	uiLenRefPosoffset			:UDINT	:= 8;
END_VAR

ACT_ReadStatus();
ACT_Power();
ACT_Jog();
ACT_Home();
IF xIsLinearMode//判断是是否是线性模式
THEN
	ACT_Move();//线性模式运动调用
ELSE
	ACT_Modulo();//模值模式调用
END_IF

ACT_Relative();
ACT_InPos();
ACT_Timeout();
ACT_Tip();
ACT_Reset();
ACT_Halt();

IF  wActionHomeStep=0 THEN
	ACT_Velocity();
	ACT_Stop();
END_IF

xPowerHmi:=FALSE;
xHomeHmi:=FALSE;
xAlarmResetHmi:=FALSE;
xPowerInit:=FALSE;
xHomeAuto:=FALSE;
//xJogForwardAuto:=FALSE;
//xJogBackwardsAuto:=FALSE;
xModulo:=FALSE;
xRelativeAuto:=FALSE;

FOR nIndex:=1 TO gc_uiAxisMoveNum DO
	//xMoveHmi[nIndex]:=FALSE;
	xMoveAuto[nIndex]:=FALSE;
END_FOR

ACTION ACT_Halt:

xHaltExecute:=xHalt;
fbHalt(
	Axis:=Axis,
	Execute:=xHaltExecute,
	Deceleration:=,
	Jerk:=,
	BufferMode:=,
	Options:=,
	Done=>,
	Busy=>,
	Active=>,
	CommandAborted=>,
	Error=>,
	ErrorID=>
);
END_ACTION

ACTION ACT_Home:

xHomeManual:=xHomeHmi
	AND xManualMode;
xHomeExecute:=xRunable
	AND (xHomeManual
		OR xHomeAuto
	);
(*fbHome(
	Axis:=Axis,
	Execute:=xHomeExecute,
	Position:=0,
	HomingMode:=iHomingMode,
	BufferMode:=,
	Options:=,
	bCalibrationCam:=xCalibrationCam,
	Done=>,
	Busy=>,
	Active=>,
	CommandAborted=>,
	Error=>,
	ErrorID=>
);*)
tHomeR_TRIG(CLK:= (*xHomeAuto  OR *) xSetPosHmi OR xHomeExecute , Q=> );
tHomeTimeOut(IN:=wActionHomeStep<>0 , PT:=T#180S , Q=> , ET=> );
IF    tHomeR_TRIG.Q THEN
	wActionHomeStep:=1;
	xHomeExecute:=FALSE;
	xQReferenceEndPosOk	:= FALSE;	
ELSIF  tHomeTimeOut.Q OR xError THEN
	wActionHomeStep:=0;
	xHomeExecute:=FALSE;
	xQReferenceEndPosOk	:= FALSE;	
END_IF
CASE wActionHomeStep OF
	(* Quickly drive in direction reference point *)
	1:  
		IF   not  xSetPosHmi  THEN
					IF xIRefSwitch THEN
						wActionHomeStep := 20;
					ELSE
						fbVelocity( Execute := FALSE, Axis := Axis );
						fbVelocity
								(	Execute		:= TRUE,
									Velocity	:= lrIRefVeloPlusFast,
									Direction	:= MC_Negative_Direction,
									Axis		:= Axis
								);
						fbVelocity( Execute := FALSE, Axis := Axis );	
					END_IF
		ELSE
			wActionHomeStep := 90;
		END_IF
	(* Stop if the reference switch is moved over *)
	10:
		IF xIRefSwitch THEN
			fbStop( Execute := FALSE, Axis := Axis );
			fbStop( Execute := TRUE, Axis := Axis );
			wActionHomeStep := 11;
		END_IF		
	11:
		IF fbStop.Busy THEN
			fbStop( Execute := FALSE, Axis := Axis );
		ELSE
			wActionHomeStep :=12;
		END_IF

	12:
		fbReferenceWait( IN := TRUE, PT := T#1000MS );
		wActionHomeStep := 13;

	13:
		fbReferenceWait();
		IF fbReferenceWait.Q THEN
			wActionHomeStep := 20;
			fbReferenceWait.IN:=FALSE;
		END_IF

	20:
		fbVelocity( Execute := FALSE, Axis := Axis );
		fbVelocity
			(	Execute		:= TRUE,
				Velocity	:= lrIRefVeloMinusFast,
				Direction	:= MC_Positive_Direction,
				Axis		:= Axis
			);
		fbVelocity( Execute := FALSE, Axis := Axis );
		IF  fbVelocity.Active   THEN
			wActionHomeStep := 30;
		END_IF
	(* Stop if the reference switch falls *)
(*	21:  
	 *)
	30:
		IF NOT xIRefSwitch THEN
			fbStop( Execute := FALSE, Axis := Axis );
			fbStop( Execute := TRUE, Axis := Axis );
			wActionHomeStep := 31;
		END_IF

	31:
		IF fbStop.Busy THEN
			fbStop( Execute := FALSE, Axis := Axis );
		ELSE
			wActionHomeStep := 32;
		END_IF

	32:
		fbReferenceWait( IN := TRUE, PT := t#100ms );
		wActionHomeStep	:= 33;

	33:
		fbReferenceWait();
		IF fbReferenceWait.Q THEN
			wActionHomeStep := 40;
			fbReferenceWait( IN := FALSE);
		END_IF
	40:
		IF xIRefSwitch THEN
			wActionHomeStep := 20;
		ELSE
		
			fbVelocity( Execute := FALSE, Axis := Axis );
			fbVelocity
				(	Execute		:= TRUE,
					Velocity	:= lrIRefVeloPlusSlow,
					Direction	:= MC_Negative_Direction,
					Axis		:= Axis
				);
			fbVelocity( Execute := FALSE, Axis := Axis );
			IF  fbVelocity.Active THEN
				wActionHomeStep := 50;
			END_IF
			
		END_IF
	(* Stop if the reference switch is moved over *)
	50:
		IF xIRefSwitch THEN
			fbStop( Execute := FALSE, Axis := Axis );
			fbStop( Execute := TRUE, Axis := Axis );
			wActionHomeStep := 51;
		END_IF

	51:
		IF fbStop.Busy THEN
			fbStop( Execute := FALSE, Axis := Axis );
		ELSE
			wActionHomeStep := 52;
		END_IF

	52:
		fbReferenceWait( IN := TRUE, PT := t#100ms );
		wActionHomeStep := 53;

	53:
		fbReferenceWait();
		IF fbReferenceWait.Q THEN
			wActionHomeStep := 60;
			fbReferenceWait( IN := FALSE);
		END_IF


	(* Slow move away from reference switch *)
	60:
		fbVelocity( Execute := FALSE, Axis := Axis );
		fbVelocity
			(	Execute		:= TRUE,
				Velocity	:= lrIRefVeloMinusSlow,
				Direction	:= MC_Positive_Direction,
				Axis		:= Axis
			);
		fbVelocity( Execute := FALSE, Axis := Axis );
		IF fbVelocity.Active THEN
				wActionHomeStep := 70;
		END_IF

	(* Stop if the reference switch falls *)
	70:
		IF NOT xIRefSwitch THEN
			fbStop( Execute := FALSE, Axis := Axis );
			fbStop( Execute := TRUE, Axis := Axis );
			wActionHomeStep := 71;
		END_IF

	71:
		IF fbStop.Busy THEN
			fbStop( Execute := FALSE, Axis := Axis );
		ELSE
			fbReferenceEndWait( IN := FALSE, PT := t#500ms );
			wActionHomeStep := 72;
		END_IF

	72:
		fbReferenceWait( IN := TRUE, PT := t#100ms );
		wActionHomeStep := 73;

	73:
		fbReferenceWait();
		IF fbReferenceWait.Q THEN
			wActionHomeStep := 80;
			fbReferenceWait( IN := FALSE);
		END_IF

	(* Wait until the position is valid *)
	80:
		fbReferenceEndWait( IN := TRUE );
		IF fbReferenceEndWait.Q THEN
				fbSetPos( Execute := FALSE, Axis := Axis );
				IF xIResetRefPosCheck THEN
					lrQReferenceCheckDiff := 0;
				ELSE
					lrQReferenceCheckDiff := lrQPositionAct - lrQReferenceEndPos;
				END_IF
			IF NOT   xIRelative_Encoder THEN
				wActionHomeStep := 90;
			ELSE	
				wActionHomeStep := 140;	
			END_IF
				
		END_IF

	90:
	
		fbAdsRead(Read:=FALSE);
		fbAdsRead(
		NETID:='' , 
		PORT:=501 , 
		IDXGRP:=NCIDXG_AXPARMS + DWORD_TO_UINT(Axis.NcToPlc.AxisId),
		IDXOFFS:=uiOffsetEncoderId, 
		LEN:= uiLenEncoderId, 
		DESTADDR:= ADR(uiencoderId),
		READ:= TRUE, 
		TMOUT:=T#1s , 
		BUSY=> , 
		ERR=> , 
		ERRID=> );
		fbAdsRead(Read:=FALSE);
		IF fbAdsRead.BUSY THEN
			fbAdsRead.READ	:= FALSE;
			wActionHomeStep  :=95;
		END_IF
	95: 
		IF	ABS(rActPos)>0.1  THEN 
			xPoweroff:=TRUE;
			IF  NOT xPowerOn THEN
				wActionHomeStep  :=100;
			END_IF
		ELSE
			wActionHomeStep  :=140;
		END_IF
	100:	
		
			rReferencePositionoffset:= -REAL_TO_LREAL(rActPos);
			fbAdsWrite(WRITE:=FALSE);
			fbAdsWrite(
					NETID:= '', 
					PORT:= 501, 
					IDXGRP:=(NCIDXG_ENCPAMS+ uiencoderId ), 
					IDXOFFS:=  uiPositionBias, 
					LEN:=  SIZEOF(rReferencePositionoffset),
					SRCADDR:= ADR(rReferencePositionoffset),
					WRITE:= TRUE, 
					TMOUT:= T#1s, 
					BUSY=> , 
					ERR=> , 
					ERRID=> );
			IF fbAdsWrite.BUSY THEN
					fbAdsWrite.WRITE	:= FALSE;
					wActionHomeStep  :=120;
			END_IF
	120:  xPoweroff:=FALSE;
		IF   xPowerOn THEN
			wActionHomeStep  :=140;
		END_IF	

	(* Set position to 0 *)
	140:
		fbSetPos( Execute := TRUE, Position :=REAL_TO_LREAL(lrIReferencePosition) , Axis := Axis );

		IF NOT fbSetPos.Busy THEN
			fbSetPos( Execute := FALSE, Axis := Axis );
			wActionHomeStep := 150;
		END_IF
	
	(* Axis set to status referenced *)
	150:	
		fbHome ( Execute := TRUE,Position:=REAL_TO_LREAL(lrIReferencePosition) ,
					HomingMode:=MC_Direct,
					bCalibrationCam:=TRUE,
 					Axis := Axis );
		IF NOT fbHome.Busy THEN
			fbHome ( Execute := FALSE, Axis := Axis );
			lrQReferenceEndPos	:= 0;
			xQReferenceEndPosOk	:= TRUE;
			wActionHomeStep		:= 0;
		END_IF
END_CASE
////正向回原---先负向（快JOG）远离DOG，在正向（慢JOG）接近DOG点。
END_ACTION

ACTION ACT_InPos:

(*FOR nIndexMove:=1 TO nMoveActualNum DO
	tonInPosition[nIndexMove](
		IN:=bReady
			AND NOT Axis.Status.Moving
			AND Axis.Status.NotMoving
			AND Axis.Status.InPositionArea
			AND Axis.Status.InTargetPosition
			AND Axis.NcToPlc.SetPos=REAL_TO_LREAL(rMovePosition[nIndexMove])
			AND Axis.NcToPlc.TargetPos=REAL_TO_LREAL(rMovePosition[nIndexMove]),
		PT:=tInPosition[nIndexMove],
		Q=>bInPosition[nIndexMove],
		ET=>
	);
END_FOR*)
//检测运行是否到位
IF xIsLinearMode THEN //线性定位
	FOR nIndexMove:=1 TO gc_uiAxisMoveNum DO
		tonInPosition[nIndexMove](
			IN:=xReady
			 AND NOT Axis.Status.Moving
			 AND Axis.Status.NotMoving
			//   AND Axis.Status.InPositionArea
			//   AND Axis.Status.InTargetPosition
			//   AND Axis.NcToPlc.SetPos=REAL_TO_LREAL(rMovePosition[nIndexMove])
			//   AND Axis.NcToPlc.TargetPos=REAL_TO_LREAL(rMovePosition[nIndexMove]),
			 AND Axis.NcToPlc.ActPos >= REAL_TO_LREAL(rMovePosition[nIndexMove] - 0.2)
			 AND Axis.NcToPlc.ActPos <= REAL_TO_LREAL(rMovePosition[nIndexMove] + 0.2),
			PT:=tInPosition[nIndexMove],
			Q=>xMoveInPos[nIndexMove],
			ET=>);
	END_FOR
ELSE//模值定位
		FOR nIndexMove:=1 TO gc_uiAxisMoveNum DO
		tonInPosition[nIndexMove](
			IN:=xReady
			 AND NOT Axis.Status.Moving
			 AND Axis.Status.NotMoving
			//   AND Axis.Status.InPositionArea
			//   AND Axis.Status.InTargetPosition
			//   AND Axis.NcToPlc.SetPos=REAL_TO_LREAL(rMovePosition[nIndexMove])
			//   AND Axis.NcToPlc.TargetPos=REAL_TO_LREAL(rMovePosition[nIndexMove]),
			 AND Axis.NcToPlc.ModuloActPos >= REAL_TO_LREAL(rMovePosition[nIndexMove] - 0.2)
			 AND Axis.NcToPlc.ModuloActPos <= REAL_TO_LREAL(rMovePosition[nIndexMove] + 0.2),
			PT:=tInPosition[nIndexMove],
			Q=>xMoveInPos[nIndexMove],
			ET=>);
	END_FOR
END_IF
END_ACTION

ACTION ACT_Jog:

xJogForwardManual:=xJogForwardHmi
	AND xManualMode;
xJogBackwardsManual:=xJogBackwardsHmi
	AND xManualMode;
xJogForward:=xRunable
	AND NOT xJogBackwards
	AND NOT xJogForwardLimit
	AND (xJogForwardManual
		OR (xJogForwardAuto AND xAutoMode)
	);
xJogBackwards:=xRunable
	AND NOT xJogForward
	AND NOT xJogBackwardsLimit
	AND (xJogBackwardsManual
		OR (xJogBackwardsAuto AND xAutoMode)
	);
fbJog(
	Axis:=Axis,
	JogForward:=xJogForward,
	JogBackwards:=xJogBackwards,
	Mode:=MC_JOGMODE_CONTINOUS,
	Position:=0,
	Velocity:=REAL_TO_LREAL(rJogVelocity),
	Acceleration:=(*REAL_TO_LREAL(rJogAcceleration)*),
	Deceleration:=(*REAL_TO_LREAL(rJogDeceleration)*),
	Jerk:=,
	Done=>,
	Busy=>,
	Active=>,
	CommandAborted=>,
	Error=>,
	ErrorID=>
);

IF NOT xAutoMode  THEN
	xJogForwardAuto:=FALSE;
	xJogBackwardsAuto:=FALSE;
	 
END_IF
END_ACTION

ACTION ACT_Modulo:
FOR nIndexMove:=1 TO gc_uiAxisMoveNum DO
	IF xAutoMode THEN
		IF rMoveVelocity[nIndexMove]>0 
		THEN
			rVelocity:=rMoveVelocity[nIndexMove];
		ELSE
			rVelocity:=rAutoVelocity;
		END_IF
	ELSE
		rVelocity:=rManualVelocity;
	END_IF	
	
	xMoveManual[nIndexMove]:=xMoveHmi[nIndexMove] AND xMoveILC[nIndexMove]
													AND xManualMode;
	xMoveExecute[nIndexMove]:=xRunable
														AND xMoveILC[nIndexMove]
														AND (xMoveManual[nIndexMove]
														OR xMoveAuto[nIndexMove]);
	fbModulo(
		Axis:=Axis,
		Execute:=xMoveExecute[nIndexMove],
		Position:=REAL_TO_LREAL(rMovePosition[nIndexMove]),
		Velocity:=REAL_TO_LREAL(rVelocity),
		Acceleration:=REAL_TO_LREAL(rMoveAcceleration),
		Deceleration:=REAL_TO_LREAL(rMoveDeceleration),
		Direction:=nModuloDirection,
		BufferMode:=,
		Options:=,
		Done=>,
		Busy=>,
		Active=>,
		CommandAborted=>,
		Error=>,
		ErrorID=>
	);
END_FOR
END_ACTION

ACTION ACT_Move:

FOR nIndexMove:=1 TO gc_uiAxisMoveNum DO
	IF xAutoMode THEN
		IF rMoveVelocity[nIndexMove]>0 
		THEN
			rVelocity:=rMoveVelocity[nIndexMove];
		ELSE
			rVelocity:=rAutoVelocity;
		END_IF
	ELSE
		rVelocity:=rManualVelocity;
	END_IF	
	
	xMoveManual[nIndexMove]:=(xMoveHmi[nIndexMove] OR xTarMoveExecute[nIndexMove])AND xMoveILC[nIndexMove]
													AND xManualMode;
	xMoveExecute[nIndexMove]:=xRunable AND xMoveILC[nIndexMove]
										AND (xMoveManual[nIndexMove]
										OR xMoveAuto[nIndexMove]);
	fbMove[nIndexMove](
		Axis:=Axis,
		Execute:=xMoveExecute[nIndexMove],
		Position:=REAL_TO_LREAL(rMovePosition[nIndexMove]),
		Velocity:=REAL_TO_LREAL(rVelocity),
		Acceleration:=REAL_TO_LREAL(rMoveAcceleration),
		Deceleration:=REAL_TO_LREAL(rMoveDeceleration),
		Jerk:=,
		BufferMode:=MC_Aborting,
		Options:=,
		Done=>xMoveDone[nIndexMove],
		Busy=>,
		Active=>,
		CommandAborted=>,
		Error=>,
		ErrorID=>
	);
END_FOR
(**********************************触摸屏中选择伺服参数************************************)
xTarMoveExecute[xITarMoveHmi]:=xITarMoveButtonHmi;
xQTarPosition			:=rMovePosition[xITarMoveHmi];
xQTarVelocity			:=rManualVelocity;
END_ACTION

ACTION ACT_Power:

rtPowerHmi(
	CLK:=xPowerHmi,
	Q=>
);
IF xEStop AND xSafety THEN
	IF rtPowerHmi.Q
		AND xKey
		AND xSafety
		AND xManualMode
	THEN
		xPowerManual:=NOT xPowerManual;
	END_IF
	IF xPowerInit THEN
		xNotPower:=FALSE;
		xPowerManual:=FALSE;
		xPowerAuto:=TRUE;
	END_IF
ELSE
	xPowerManual:=FALSE;
	xPowerAuto:=FALSE;
END_IF
xPowerEnable:=NOT Axis.Status.Error
						AND (xPowerManual XOR xPowerAuto);
fbPower(
	Axis:=Axis,
	Enable:=xPowerEnable AND NOT xSv_not_power AND NOT xNotPower AND  NOT xPoweroff,
	Enable_Positive:=xEnablePositive,
	Enable_Negative:=xEnableNegative,
	Override:=100,
	BufferMode:=,
	Options:=,
	Status=>xPowerOn,
	Busy=>,
	Active=>,
	Error=>,
	ErrorID=>
);
//xPowerOn := Axis.NcToPlc.StateDWord.1;
//Axis.Status;
//AXIS.NcToPlc.StateDWord;
//AXIS.NcToPlc.StateDWord2;
//AXIS.NcToPlc.StateDWord3;
uiStatusCopy[2].1;
uiStatusCopy[2];
xReady:=xPowerOn
	AND NOT Axis.Status.Error
	AND Axis.Status.Operational;
xRunable:=xEStop
	AND xKey
	AND xSafety
	AND xReady
	AND xRunILC;
END_ACTION

ACTION ACT_ReadStatus:

fbReadStatus(
	Axis:=Axis,
	Enable:=TRUE,
	Valid=>,
	Busy=>,
	Error=>,
	ErrorID=>,
	ErrorStop=>,
	Disabled=>,
	Stopping=>,
	StandStill=>,
	DiscreteMotion=>,
	ContinuousMotion=>,
	SynchronizedMotion=>,
	Homing=>,
	ConstantVelocity=>,
	Accelerating=>,
	Decelerating=>,
	Status=>
);

xError					:=Axis.Status.Error;
nErrorID				:=Axis.Status.ErrorID;
xbusy					:=Axis.Status.Moving;
nErrorCode				:=Axis.NcToPlc.ErrorCode;


rSetTorque				:=LREAL_TO_REAL(Axis.NcToPlc.SetTorque);
rSetPos					:=LREAL_TO_REAL(Axis.NcToPlc.SetPos);
rModuloSetPos			:=LREAL_TO_REAL(Axis.NcToPlc.ModuloSetPos);
rModuloSetTurns			:=LREAL_TO_REAL(Axis.NcToPlc.ModuloSetTurns);
rTargetPos				:=LREAL_TO_REAL(Axis.NcToPlc.TargetPos);

rActTorque				:=LREAL_TO_REAL(Axis.NcToPlc.ActTorque);
IF xIsLinearMode//判断是是否是线性模式(不同模式读取的数据源不同)
THEN
	rActPos					:=LREAL_TO_REAL(Axis.NcToPlc.ActPos);
ELSE
	rActPos			    :=LREAL_TO_REAL(Axis.NcToPlc.ModuloActPos);
END_IF
rActVelo				:=LREAL_TO_REAL(Axis.NcToPlc.ActVelo);

rPosDiff				:=LREAL_TO_REAL(Axis.NcToPlc.PosDiff);

NcToPlc					:=Axis.NcToPlc;
Status					:=Axis.Status;
END_ACTION

ACTION ACT_Relative:
IF xAutoMode THEN
	IF rRelativeVelocity>0 THEN
		rVelocity:=rRelativeVelocity;
	ELSE
		rVelocity:=rAutoVelocity;
	END_IF
ELSE
	rVelocity:=rManualVelocity;
END_IF
xRelativeExecute:=xRunable
		AND ((xRelativeHmi AND xManualMode) OR xRelativeAuto (*AND xAutoMode*)) AND xRelativeILC;

fbRelative(
	Axis:=Axis,  
	Execute:= xRelativeExecute, 
	Distance:= REAL_TO_LREAL(rRelativeDistance), 
	Velocity:= REAL_TO_LREAL(rVelocity), 
	Acceleration:= rMoveAcceleration, 
	Deceleration:= rMoveDeceleration, 
	Jerk:= , 
	Done=> xRelativeDone, 
	Busy=> xRelativeBusy, 
	CommandAborted=> , 
	Error=> xRelativeError, 
	ErrorID=> udiRelativeErrorID);
	
IF xRelativeDone=TRUE THEN
	xRelativeDone1:=TRUE;
ELSIF xRelativeBusy=TRUE THEN
	xRelativeDone1:=FALSE;	
END_IF//
END_ACTION

ACTION ACT_Reset:
xResetExecute:=xAlarmReset
	OR xAlarmResetHmi;
	
fbReset(
	Axis:=Axis,
	Execute:=xResetExecute AND ( Axis.Status.Error OR NOT xPowerOn) ,
	Done=>,
	Busy=>,
	Error=>,
	ErrorID=>
);
END_ACTION

ACTION ACT_Stop:

xStopExecute:=xStop OR (xStopHmi AND xManualMode);
fbStop(
	Axis:=Axis,
	Execute:=xStopExecute,
	Deceleration:=,
	Jerk:=,
	Options:=,
	Done=>,
	Busy=>,
	Active=>,
	CommandAborted=>,
	Error=>,
	ErrorID=>
);
END_ACTION

ACTION ACT_Timeout:

IF xResetExecute THEN
	xMoveTimeout:=FALSE;
END_IF

IF NOT xMoveTimeout THEN
	FOR nIndexMove:=1 TO gc_uiAxisMoveNum DO
		tonMoveTimeout[nIndexMove](
			IN:=xMoveAuto[nIndexMove],
			PT:=tMoveTimeout,
			Q=>, ET=>
		);
		IF tonMoveTimeout[nIndexMove].Q THEN
			xMoveTimeout:=TRUE;
			EXIT;
		END_IF
	END_FOR
END_IF
END_ACTION

ACTION ACT_Tip:

IF xResetExecute THEN
	wManualTip:=0;
	xNotPowerOn:=FALSE;
END_IF

IF NOT (xPowerManual XOR xPowerAuto) 
	AND xAutoMode
	AND NOT Axis.Status.Error
THEN
	xNotPowerOn:=TRUE;
END_IF
END_ACTION

ACTION ACT_Velocity:
IF xAutoMode THEN
	IF rVelocityVel>0 THEN
		fbVelocity.Velocity:=rVelocityVel;
	ELSE
		fbVelocity.Velocity:=rAutoVelocity;
	END_IF
ELSE
	fbVelocity.Velocity:=rManualVelocity;
END_IF
xVelocityExecute:=xRunable AND xVelocityAuto AND xVelocityILC;

fbVelocity(
	Axis:=Axis , 
	Execute:=xVelocityExecute AND xVelocityAble , 
	Velocity:= , 
	Acceleration:=rVelocityAcc , 
	Deceleration:=rVelocityDec , 
	Jerk:= , 
	Direction:= , 
	InVelocity=>xVelocityInVel , 
	Busy=>xVelocityBusy , 
	CommandAborted=> , 
	Error=>xVelocityError , 
	ErrorID=>udiVelocityErrorID );
	
xVelocityAble:= NOT xVelocityAble;
END_ACTION

END_FUNCTION_BLOCK

// ---- POUs/003_FB/Z_ERG_20 FB/FB_ERG_20_Modbus.TcPOU
FUNCTION_BLOCK FB_ERG_20_Modbus//慧琳夹爪旋转模块程序
VAR_INPUT
	xExecute: BOOL;
	xAbort: BOOL;
	xResetRequest: BOOL;//匹配复位按钮 
	xPowerHmi: BOOL:=true;////上电信号，反转型
	dwTimeLimit: DWORD:=1;//[ms],1 => no invocation time limit
	dwTimeOut: DWORD;//[ms],0 => no executing time limit
	stPara       : ST_ERG_20_Sys_Para;//系统参数	
	//手动执行部分
	xHMInitButton , xInitControl : BOOL;
	aHMIClampButton , aHMIReleaseButton , aClampControl , aReleaseControl : ARRAY[1..5] OF BOOL;//手动和自动部分控制
	aHMIRotateClampButton , aHMIRotateReleaseButton , aRotateClampControl , aRotateReleaseControl : ARRAY[1..5] OF BOOL;//手动和自动部分控制
	aHMIRotateClampRelButton , aHMIRotateReleaseRelButton , aRotateClampRelControl , aRotateReleaseRelControl : ARRAY[1..5] OF BOOL;//手动和自动部分控制
	aHMIClampPara , aHMIReleasePara : ARRAY[1..5] OF ST_Huiling_PosPara;//夹紧轴点位信息
	aHMIRotateClampPara , aHMIRotateReleasePara : ARRAY[1..5] OF ST_Huiling_PosPara;//旋转轴点位信息
	aHMIRotateClampRelPara , aHMIRotateReleaseRelPara : ARRAY[1..5] OF ST_Huiling_PosPara;//旋转轴点位信息
	xAutoMode    : BOOL;//0:mannal 1:auto
	xDeviceRunning     : BOOL;//流程运行过程中
	xIniting : BOOL;
END_VAR
VAR_OUTPUT
	xDone: BOOL;(*完成条件满足*)
	xBusy: BOOL;(*动作正在执行*)
	xAborted: BOOL;(*指令被打断*)
	xError: BOOL;(*错误条件满足*)
	eErrorID: ERG_20_ERROR;(*错误码*)
	xRdyCmd : BOOL;
	xRefOk    : BOOL;    
	xGripClampEmpty : BOOL;//夹爪夹空
	xClosecoverFailure : BOOL;
	xOpencoverFailure : BOOL;
	xDropOccur : BOOL;//掉落发生
	sHmiError	: STRING;
 	eCommErrorID: BYTE;
	eOperErrorID: DWORD;
END_VAR
VAR_IN_OUT
	st_IOData : ST_ERG_20_IOData;
END_VAR
VAR
	//指令触发
	_xDone: BOOL;
	_rIniting : Tc2_Standard.R_TRIG;
	eCmd         : ERG_20_CMD;
	eClampActCmd : ERG_20_CMD;	
	rTorqueSet   : REAL;//目标力值设置
	rSpeedSet    : REAL;;//运行速度设置
	rPosAngleSet : REAL;//位置和速度设置值	
	eState: STATE;//device当前状态	
	xFirstInvocation: BOOL := TRUE;	 
	xTimeOut: BOOL;
	tOperationTimer : TON;
	_tonTimeout , _tonCmdTimeout ,_tonPulse , _tonDelay , _tonDelay1 , _tonDelay2 , _tonDelay3: TON;	
  /// detect rising edge of command execution 
	_diCmdState 	: DINT;  
	i, ii , _idx : INT;
	_xConnectError : BOOL;
	_iComNGCount : INT;
	_fResetCheck : F_TRIG;
	_fManual : F_TRIG;
	_rManual : R_TRIG;	
	_fPowerOn : F_TRIG;
	_rHMIInit , _rInit: R_TRIG;//初始化指令触发
	_rHMIClamp , _rHMIRelease , _rClamp , _rRelease : ARRAY[1..5] OF R_TRIG;//夹紧轴指令触发
	_rHMIRotateClamp , _rHMIRotateRelease , _rRotateClamp , _rRotateRelease : ARRAY[1..5] OF R_TRIG;//旋转轴指令触发
	_rHMIRotateRelClamp , _rHMIRotateRelRelease , _rRotateRelClamp , _rRotateRelRelease : ARRAY[1..5] OF R_TRIG;//旋转轴指令触发
	_iConnectState : INT := 0;//
	_connectTon : TON;

	_aRead_VAR: FB_MBReadRegs;;			//0:状态反馈数据(16#40)
	_aWtirt_VAR: ARRAY[0..3] OF FB_MBWriteRegs;	    //0:初始化控制(16#0);1:夹紧控制(16#2);2:旋转绝对定位控制(16#A);3:相对旋转
	_iSendReceiveState : INT := 0;//发送状态标志位
	_aEnableSignal : ARRAY[0..4] OF BOOL;//0:初始化控制；1:夹紧控制；2:旋转绝对定位控制;3:相对旋转; 4:状态反馈	
	_iChannelIndex:INT;
	_wPosSetTemp , _wSpeedSetTemp , _wForseSetTemp : WORD;
	_wPosSetTemp1 , _wSpeedSetTemp1 , _wForseSetTemp1 : WORD;
	_wPosSetTemp2 , _wSpeedSetTemp2 , _wForseSetTemp2 : WORD;
		
	_aReadDataTemp , _aReadDataTemp1 : ARRAY[0..5] OF INT;//夹持和旋转数据缓存
	_aFeedbackData: ARRAY[0..17] OF INT;
	_aControlData: ARRAY[0..3, 0..7] OF INT;
	_xConnect_ERROR : BOOL;
	_xModeChange : BOOL;
	_xReadStatus : BOOL := TRUE;//上电是默认读取模式的
	_iCount : INT := 0;	
	_iNGCount : INT;	
	_xBusy : BOOL;
	_xHMIOpe,_xAutoOpe : BOOL;
	_rAcceleration : REAL:=5000;
	_rTempAcceleration : REAL;
	_rLastRotatePos : REAL;
	diOldStep:DINT;
END_VAR
VAR_TEMP
	xAgain: BOOL;
END_VAR

xAgain:=0;
ConnectAction();//触发通信连接功能连接
ACTMap();//数据映射
IF eState<>STATE.DORMANT
THEN
	_rHMIInit(CLK:=FALSE) ;
	_rInit(CLK:=FALSE) ;
	FOR ii :=1 TO 5 DO
		 _rHMIClamp[ii](CLK:=FALSE);
		 _rHMIRelease[ii](CLK:=FALSE);
		 _rClamp[ii](CLK:=FALSE);
		 _rRelease[ii](CLK:=FALSE);
		 _rHMIRotateClamp[ii](CLK:=FALSE);
		 _rHMIRotateRelease[ii](CLK:=FALSE);
		 _rRotateClamp[ii](CLK:=FALSE);
		 _rRotateRelease[ii](CLK:=FALSE);
		 _rHMIRotateRelClamp[ii](CLK:=FALSE);
		 _rHMIRotateRelRelease[ii](CLK:=FALSE);
		 _rRotateRelClamp[ii](CLK:=FALSE);
		 _rRotateRelRelease[ii](CLK:=FALSE);
	END_FOR
END_IF

REPEAT
	CASE eState OF
		STATE.DORMANT:
			HandleDormantState(xAgain=> xAgain);
		STATE.EXECUTING:
			HandleExecutingState(xAgain=> xAgain);
		STATE.DONE:
			HandleDoneState(xAgain=> xAgain);
		STATE.INERROR:
			HandleErrorState(xAgain=> xAgain);
		STATE.ABORTING:
			HandleAbortingState(xAgain=> xAgain);
		STATE.ABORTED:
			HandleAbortedState(xAgain=> xAgain);
		STATE.RESETING:
			HandleResettingState(xAgain=> xAgain);
	END_CASE
UNTIL (xAgain=0)
END_REPEAT
	
CASE eErrorID OF
	ERG_20_ERROR.NO_ERROR:
		sHmiError:='NO_ERROR';	
  ERG_20_ERROR.FLT_PARA:
		sHmiError:='FLT_PARA';	
  ERG_20_ERROR.FLT_CONNECT:
		sHmiError:='FLT_CONNECT';	
  ERG_20_ERROR.FLT_RDYCMD:
		sHmiError:='FLT_RDYCMD';	
	ERG_20_ERROR.FLT_DEVICE_ERROR:
		sHmiError:='FLT_DEVICE_ERROR';	
	ERG_20_ERROR.FLT_POWERON:
		sHmiError:='FLT_POWERON';
  ERG_20_ERROR.FLT_CLAMP_TIMEOUT:
		sHmiError:='FLT_CLAMP_TIMEOUT';
  ERG_20_ERROR.FLT_ROTATE_TIMEOUT:
		sHmiError:='FLT_ROTATE_TIMEOUT';
  ERG_20_ERROR.FLT_ORG_TIMEOUT:
		sHmiError:='FLT_ORG_TIMEOUT';
	ERG_20_ERROR.FLT_CLAMPCMD_TIMEOUT:
		sHmiError:='FLT_CLAMPCMD_TIMEOUT';
  ERG_20_ERROR.FLT_ROTATECMD_TIMEOUT:
		sHmiError:='FLT_ROTATECMD_TIMEOUT';
  ERG_20_ERROR.FLT_ORGCMD_TIMEOUT:
		sHmiError:='FLT_ORGCMD_TIMEOUT';
	ERG_20_ERROR.FLT_CLAMP_DROP:
		sHmiError:='FLT_CLAMP_DROP';  
  ERG_20_ERROR.FLT_xRefOk:
		sHmiError:='FLT_xRefOk';  
	ERG_20_ERROR.FLT_CLAMP_PARA:
		sHmiError:='FLT_CLAMP_PARA'; 		
	ERG_20_ERROR.FLT_ClAMP_RELEASEFAIL:
		sHmiError:='FLT_ClAMP_RELEASEFAIL';	
  ERG_20_ERROR.FLT_ClAMP_CLAMPFAIL:
		sHmiError:='FLT_ClAMP_CLAMPFAIL';	
	ERG_20_ERROR.FLT_ROTATE_CLAMPFAIL:
		sHmiError:='FLT_ROTATE_CLAMPFAIL';	
	ERG_20_ERROR.FLT_ROTATE_RELEASEFAIL:
		sHmiError:='FLT_ROTATE_RELEASEFAIL';	
END_CASE

//检测是否有手动操作
_xHMIOpe := xHMInitButton;
FOR i := 1 TO 5 BY 1
DO
	_xHMIOpe := _xHMIOpe OR aHMIClampButton[i] OR aHMIReleaseButton[i] OR aHMIRotateClampButton[i] OR aHMIRotateClampRelButton[i] 
							OR aHMIRotateReleaseButton[i] OR aHMIRotateReleaseReLButton[i];
END_FOR

//检测是否有自动操作指令
_xAutoOpe := xInitControl;
FOR i := 1 TO 5 BY 1
DO
	_xAutoOpe := _xAutoOpe OR aClampControl[i] OR aReleaseControl[i] OR aRotateClampControl[i] OR aRotateClampRelControl[i] 
							OR aRotateReleaseControl[i] OR aRotateReleaseRelControl[i];
END_FOR

{attribute 'hide'}
METHOD AbortAction
VAR_INPUT
END_VAR
VAR_OUTPUT
	xComplete: BOOL;
  eErrorID: ERG_20_ERROR;
END_VAR
(*
* Cleaning
* => abort all running operation
* => if an NBS.ERROR codition is reached, set eErrorID to a Value rather then NBS.ERG_20_ERROR.NO_ERROR 
*)
(*
* Cleaning
* => abort all running operation
* => if an NBS.JD_EPG30_050_ERROR codition is reached, set eERRORID to a Value rather then NBS.JD_EPG30_050_ERROR.NO_ERROR 
*)
xComplete:=1;
eERRORID:=ERG_20_ERROR.NO_ERROR;
END_METHOD

ACTION ACTMap:
//进行数据映射的前提条件是外部所配置的参数是没有问题的
IF TRUE
THEN
	//进行输入数据刷新
	st_IOData.I_ClampInit := _aFeedbackData[0];
	st_IOData.I_ClampState := _aFeedbackData[1];
	//夹持信息
	_aReadDataTemp[0] := _aFeedbackData[3];
	_aReadDataTemp[1] := _aFeedbackData[2];
	_aReadDataTemp[2] := _aFeedbackData[5];
	_aReadDataTemp[3] := _aFeedbackData[4];
	_aReadDataTemp[4] := _aFeedbackData[7];
	_aReadDataTemp[5] := _aFeedbackData[6];
	
	SysMemCpy(ADR(st_IOData.I_ClampCurrentPos),ADR(_aReadDataTemp[0]),4);
	SysMemCpy(ADR(st_IOData.I_ClampCurrentSpeed),ADR(_aReadDataTemp[2]),4);
	SysMemCpy(ADR(st_IOData.I_ClampCurrentForce),ADR(_aReadDataTemp[4]),4);	
	//旋转信息
	st_IOData.I_RotateState := _aFeedbackData[8];
	
	_aReadDataTemp1[0] := _aFeedbackData[11];
	_aReadDataTemp1[1] := _aFeedbackData[10];
	_aReadDataTemp1[2] := _aFeedbackData[13];
	_aReadDataTemp1[3] := _aFeedbackData[12];
	_aReadDataTemp1[4] := _aFeedbackData[15];
	_aReadDataTemp1[5] := _aFeedbackData[14];
	
	SysMemCpy(ADR(st_IOData.I_RotateCurrentPos),ADR(_aReadDataTemp1[0]),4);
	SysMemCpy(ADR(st_IOData.I_RotateCurrentSpeed),ADR(_aReadDataTemp1[2]),4);
	SysMemCpy(ADR(st_IOData.I_RotateCurrentForce),ADR(_aReadDataTemp1[4]),4);	

	//进行输出数据刷新(外面一定要用保持性的数据来定义)	
	_aControlData[0,0] := st_IOData.O_Init;
	
	SysMemCpy(ADR(_aControlData[1,0]),ADR(st_IOData.O_ClampPosSet),4);//夹持位置设定	
	//进行高低位的互换
	_wPosSetTemp := TO_WORD(_aControlData[1,0]);
	_aControlData[1,0] := _aControlData[1,1];
	_aControlData[1,1] := TO_INT(_wPosSetTemp);
	
	SysMemCpy(ADR(_aControlData[1,2]),ADR(st_IOData.O_ClampSpeedSet),4);//夹持速度设定
	//进行高低位的互换
	_wSpeedSetTemp := TO_WORD(_aControlData[1,2]);
	_aControlData[1,2] := _aControlData[1,3];
	_aControlData[1,3] := TO_INT(_wSpeedSetTemp);
	//晶晶
	SysMemCpy(ADR(_aControlData[1,4]),ADR(st_IOData.O_ClampForceSet),4);//夹持力矩设定	
	//进行高低位的互换
	_wForseSetTemp := TO_WORD(_aControlData[1,4]);
	_aControlData[1,4] := _aControlData[1,5];
	_aControlData[1,5] := TO_INT(_wForseSetTemp);	
	(************************************旋转输出控制**********************************)
		//旋转绝对定位
	IF eCmd = ERG_20_CMD.Cmd_RotateAbsClamp OR eCmd = ERG_20_CMD.Cmd_RotateAbsRelease
	THEN
		SysMemCpy(ADR(_aControlData[2,0]),ADR(st_IOData.O_RotatePosSet),4);//旋转角度设定	
		//进行高低位的互换
		_wPosSetTemp1 := TO_WORD(_aControlData[2,0]);
		_aControlData[2,0] := _aControlData[2,1];
		_aControlData[2,1] := TO_INT(_wPosSetTemp1);
		
		SysMemCpy(ADR(_aControlData[2,4]),ADR(st_IOData.O_RotateSpeedSet),4);//旋转速度设定
		//进行高低位的互换
		_wSpeedSetTemp1 := TO_WORD(_aControlData[2,4]);
		_aControlData[2,4] := _aControlData[2,5];
		_aControlData[2,5] := TO_INT(_wSpeedSetTemp1);
		
		//晶晶
		SysMemCpy(ADR(_aControlData[2,6]),ADR(st_IOData.O_RotateForceSet),4);//旋转电流设定
		//进行高低位的互换
		_wForseSetTemp1 := TO_WORD(_aControlData[2,6]);
		_aControlData[2,6] := _aControlData[2,7];
		_aControlData[2,7] := TO_INT(_wForseSetTemp1);
	END_IF
	//旋转相对定位
	IF eCmd = ERG_20_CMD.Cmd_RotateRelClamp OR eCmd = ERG_20_CMD.Cmd_RotateRelRelease
	THEN		
		SysMemCpy(ADR(_aControlData[3,0]),ADR(st_IOData.O_RotateSpeedSet),4);//旋转速度设定
		//进行高低位的互换
		_wSpeedSetTemp2 := TO_WORD(_aControlData[3,0]);
		_aControlData[3,0] := _aControlData[3,1];
		_aControlData[3,1] := TO_INT(_wSpeedSetTemp2);
		//晶晶
		SysMemCpy(ADR(_aControlData[3,2]),ADR(st_IOData.O_RotateForceSet),4);//旋转电流设定
		//进行高低位的互换
		_wForseSetTemp2 := TO_WORD(_aControlData[3,2]);
		_aControlData[3,2] := _aControlData[3,3];
		_aControlData[3,3] := TO_INT(_wForseSetTemp2);		

		_rAcceleration:= 5000;
		SysMemCpy(ADR(_aControlData[3,4]),ADR(_rAcceleration),4);//加速度
		//进行高低位的互换
		_rTempAcceleration := TO_WORD(_aControlData[3,4]);
		_aControlData[3,4] := _aControlData[3,5];
		_aControlData[3,5] := TO_INT(_rTempAcceleration);		
		
		SysMemCpy(ADR(_aControlData[3,6]),ADR(st_IOData.O_RotatePosSet),4);//旋转角度设定	
		//进行高低位的互换
		_wPosSetTemp2 := TO_WORD(_aControlData[3,6]);
		_aControlData[3,6] := _aControlData[3,7];
		_aControlData[3,7] := TO_INT(_wPosSetTemp2);		
		
	END_IF	
	
END_IF
_rIniting(CLK:= xIniting);//检测是否是初始化中，如果是的去切换模式
IF _rIniting.Q
THEN
	eState := STATE.RESETING;
END_IF
_fResetCheck(CLK:=xResetRequest);
xRdyCmd := xPowerHmi AND(( eState = STATE.DORMANT ) OR (NOT xAutoMode AND _xAutoOpe AND eState = STATE.DONE ));//检测是否允许指令控制
//检测是否有模式变化
_fManual(CLK:=xAutoMode);
_rManual(CLK:=xAutoMode);
IF eState <> STATE.DORMANT//只有在运行的时候，才会检测是否有模式切换发生
THEN
	IF _fManual.Q OR _rManual.Q
	THEN
		_xModeChange := TRUE;
	END_IF
END_IF

_tonPulse(IN:=NOT _tonPulse.Q , PT:=T#100MS);//产生100ms的脉冲信号
IF _xReadStatus AND ( _iSendReceiveState <> 999 ) AND TRUE//一定要处于通信正常状态
THEN
		_aRead_VAR.bExecute := _tonPulse.Q;
END_IF

(****************************电源控制********************************************)

_fPowerOn(CLK:= xPowerHmi);//驱动器断电的时候需要将初始化完成信号给清除掉
IF _fPowerOn.Q
THEN
	xRefOk := FALSE;//断电再上电之后需要重新初始化
END_IF

(*****************************夹爪状态显示*****************************)
xDone := _xDone AND xExecute;//判断是否处于当前流程的Done状态
xDropOccur :=( eClampActCmd = ERG_20_CMD.Cmd_Clamp ) AND ( st_IOData.I_ClampState = 3 );
xGripClampEmpty := xError AND eErrorID = ERG_20_ERROR.FLT_ClAMP_CLAMPFAIL AND xExecute;//关盖失败判定
xClosecoverFailure := xError AND eErrorID = ERG_20_ERROR.FLT_ROTATE_CLAMPFAIL AND xExecute;//关盖失败判定
xOpencoverFailure := xError AND eErrorID = ERG_20_ERROR.FLT_ROTATE_RELEASEFAIL AND xExecute;//开盖失败评定
END_ACTION

METHOD CmdClampAction
VAR_OUTPUT
	xComplete: BOOL;
END_VAR
// return the real actual fault number
IF eErrorID <> ERG_20_ERROR.NO_ERROR
THEN
  RETURN;  
END_IF
  
IF NOT xRefOk THEN
	eErrorID := ERG_20_ERROR.FLT_xRefOk;
	RETURN;
END_IF

IF rTorqueSet>0.5 OR rTorqueSet<0.1
	OR rSpeedSet>400 OR rSpeedSet<1
	OR rPosAngleSet>20 OR rPosAngleSet<0
THEN
	eErrorID := ERG_20_ERROR.FLT_PARA;	
END_IF

